//   XtsTransport/XtsTransport Instance <-> NC-Task 1/Axes/Mover Axis 86
//     PlcTask Inputs/GVL_XTS.AxisRefMover[86].NcToPlc <-> Outputs/ToPlc
//     PlcTask Outputs/GVL_XTS.AxisRefMover[86].PlcToNc <-> Inputs/FromPlc
//   XtsTransport/XtsTransport Instance <-> NC-Task 1/Axes/Mover Axis 87
//     PlcTask Inputs/GVL_XTS.AxisRefMover[87].NcToPlc <-> Outputs/ToPlc
//     PlcTask Outputs/GVL_XTS.AxisRefMover[87].PlcToNc <-> Inputs/FromPlc
//   XtsTransport/XtsTransport Instance <-> NC-Task 1/Axes/Mover Axis 88
//     PlcTask Inputs/GVL_XTS.AxisRefMover[88].NcToPlc <-> Outputs/ToPlc
//     PlcTask Outputs/GVL_XTS.AxisRefMover[88].PlcToNc <-> Inputs/FromPlc
//   XtsTransport/XtsTransport Instance <-> NC-Task 1/Axes/Mover Axis 89
//     PlcTask Inputs/GVL_XTS.AxisRefMover[89].NcToPlc <-> Outputs/ToPlc
//     PlcTask Outputs/GVL_XTS.AxisRefMover[89].PlcToNc <-> Inputs/FromPlc
//   XtsTransport/XtsTransport Instance <-> NC-Task 1/Axes/Mover Axis 9
//     PlcTask Inputs/GVL_XTS.AxisRefMover[9].NcToPlc <-> Outputs/ToPlc
//     PlcTask Outputs/GVL_XTS.AxisRefMover[9].PlcToNc <-> Inputs/FromPlc
//   XtsTransport/XtsTransport Instance <-> NC-Task 1/Axes/Mover Axis 90
//     PlcTask Inputs/GVL_XTS.AxisRefMover[90].NcToPlc <-> Outputs/ToPlc
//     PlcTask Outputs/GVL_XTS.AxisRefMover[90].PlcToNc <-> Inputs/FromPlc
//   XtsTransport/XtsTransport Instance <-> NC-Task 1/Axes/Mover Axis 91
//     PlcTask Inputs/GVL_XTS.AxisRefMover[91].NcToPlc <-> Outputs/ToPlc
//     PlcTask Outputs/GVL_XTS.AxisRefMover[91].PlcToNc <-> Inputs/FromPlc
//   XtsTransport/XtsTransport Instance <-> NC-Task 1/Axes/Mover Axis 92
//     PlcTask Inputs/GVL_XTS.AxisRefMover[92].NcToPlc <-> Outputs/ToPlc
//     PlcTask Outputs/GVL_XTS.AxisRefMover[92].PlcToNc <-> Inputs/FromPlc
//   XtsTransport/XtsTransport Instance <-> NC-Task 1/Axes/Mover Axis 93
//     PlcTask Inputs/GVL_XTS.AxisRefMover[93].NcToPlc <-> Outputs/ToPlc
//     PlcTask Outputs/GVL_XTS.AxisRefMover[93].PlcToNc <-> Inputs/FromPlc
//   XtsTransport/XtsTransport Instance <-> NC-Task 1/Axes/Mover Axis 94
//     PlcTask Inputs/GVL_XTS.AxisRefMover[94].NcToPlc <-> Outputs/ToPlc
//     PlcTask Outputs/GVL_XTS.AxisRefMover[94].PlcToNc <-> Inputs/FromPlc
//   XtsTransport/XtsTransport Instance <-> NC-Task 1/Axes/Mover Axis 95
//     PlcTask Inputs/GVL_XTS.AxisRefMover[95].NcToPlc <-> Outputs/ToPlc
//     PlcTask Outputs/GVL_XTS.AxisRefMover[95].PlcToNc <-> Inputs/FromPlc
//   XtsTransport/XtsTransport Instance <-> NC-Task 1/Axes/Mover Axis 96
//     PlcTask Inputs/GVL_XTS.AxisRefMover[96].NcToPlc <-> Outputs/ToPlc
//     PlcTask Outputs/GVL_XTS.AxisRefMover[96].PlcToNc <-> Inputs/FromPlc
//   XtsTransport/XtsTransport Instance <-> NC-Task 1/Axes/Mover Axis 97
//     PlcTask Inputs/GVL_XTS.AxisRefMover[97].NcToPlc <-> Outputs/ToPlc
//     PlcTask Outputs/GVL_XTS.AxisRefMover[97].PlcToNc <-> Inputs/FromPlc
//   XtsTransport/XtsTransport Instance <-> NC-Task 1/Axes/Mover Axis 98
//     PlcTask Inputs/GVL_XTS.AxisRefMover[98].NcToPlc <-> Outputs/ToPlc
//     PlcTask Outputs/GVL_XTS.AxisRefMover[98].PlcToNc <-> Inputs/FromPlc
//   XtsTransport/XtsTransport Instance <-> NC-Task 1/Axes/Mover Axis 99
//     PlcTask Inputs/GVL_XTS.AxisRefMover[99].NcToPlc <-> Outputs/ToPlc
//     PlcTask Outputs/GVL_XTS.AxisRefMover[99].PlcToNc <-> Inputs/FromPlc
//   XtsTransport/XtsTransport Instance <-> NC-Task 1/Objects/Group1 (CA Group)
//     PlcTask Inputs/GVL_XTS.CaGroupRef.NcToPlc/CA <-> Group Outputs/ToPLC
//     PlcTask Outputs/GVL_XTS.CaGroupRef.PlcToNc/CA <-> Group Inputs/FromPLC

// ---- APPLICATION/_types/E_PROCESS_CTRL.TcDUT
{attribute 'qualified_only'}
{attribute 'strict'}
{attribute 'to_string'}
TYPE E_PROCESS_CTRL :
(
  PROCESS_INIT              := 10,
  PROCESS_DISABLE           := 20,
  PROCESS_ENABLE            := 30,

  PROCESS_STATIONS_ENTER    := 40,
  PROCESS_STATIONS_SEND,

  PROCESS_START             := 60,
  PROCESS_DONE              := 70,
  PROCESS_STATIONS_OUTFEED  := 80
);
END_TYPE

// ---- APPLICATION/_types/LinkedList/ST_PROCESS_LIST_RESULT.TcDUT
TYPE ST_PROCESS_LIST_RESULT :
STRUCT
  wState    : WORD;   // wState == 0 --> all ok
  nIndex    : ULINT;
  stData    : ST_PROCESS_DATA;  // copy of list entry
END_STRUCT
END_TYPE

// ---- MAPPING/_types/U_APP_CTRL.TcDUT
TYPE U_APP_CTRL :
UNION
  stCtrl              : ST_APP_CTRL;
  byCtrl    AT %Q*    : ARRAY[1..SIZEOF(ST_APP_CTRL)] OF BYTE;
END_UNION
END_TYPE

// ---- XTS_TRANSPORT/XtsStation/types/E_STATION_GEAR_DISTANCE_AXIS.TcDUT
{attribute 'qualified_only'}
{attribute 'strict'}
{attribute 'to_string'}
TYPE E_STATION_GEAR_DISTANCE_AXIS :
(
  // which axis nSync distance is checked for termination of GearInPosCA.
  // after nSync distance the station does a regular outfeed to target station
	FOLLOW_THE_MASTER,
  FOLLOW_THE_SLAVE
)UINT;
END_TYPE

// ---- _MSG/types/ST_MESSAGE_STATE.TcDUT
TYPE ST_MESSAGE_STATE :
STRUCT
  State         : E_MESSAGE_STATE;  // as always... combined value of Cmd equivalent and e_progress
END_STRUCT
END_TYPE

// ---- APPLICATION/GVL_APPLICATION.TcGVL
VAR_GLOBAL CONSTANT
  MAX_PROCESS       : UINT := 20;
END_VAR
{attribute 'qualified_only'}
VAR_GLOBAL
  Simulation        : ARRAY[1..MAX_PROCESS] OF fb_Simulation;
END_VAR

// ---- XTS_TRANSPORT/GVL_XTS_CONSTANTS.TcGVL
//{attribute 'qualified_only'}
VAR_GLOBAL CONSTANT
//-----------------------------------------------------------------------------------------------------------------------------------------
//-----------------------------------------------------------------------------------------------------------------------------------------
//
//  HAUD 2026.03.15
//  - parameter list deleted (never used the parameter feature anyway), 
//    back to static global constants
//
//-----------------------------------------------------------------------------------------------------------------------------------------
//-----------------------------------------------------------------------------------------------------------------------------------------
//  Connections to XTS Utility Lib data: 
//  - suits this simple approach, 
//  - leaves you options to expand, 
//  - expansion and multiplication is not implemented here on purpose, 
//  - this project is designed to get the main ideas across, 
//  - setting up a matrix for multiple fb_Xpu instances with it, 
//    --> a second step you might want to organize from here; 
//        --> I leave the details up to you
//-----------------------------------------------------------------------------------------------------------------------------------------
//-----------------------------------------------------------------------------------------------------------------------------------------
  MAX_MOVER             : UINT    := 108;
//   MAX_MOVER           : UINT    := TO_UINT(Tc3_XTS_Utility.TcIoXtsEnvironmentParameterList.MaxXtsMoversPerXpu);
//   MAX_MODULE          : UINT    := TO_UINT(Tc3_XTS_Utility.TcIoXtsEnvironmentParameterList.MaxModulesPerPart);
//   MAX_PART            : UINT    := TO_UINT(Tc3_XTS_Utility.TcIoXtsEnvironmentParameterList.MaxXtsPartsPerXpu);
//   MAX_TRACK           : UINT    := TO_UINT(Tc3_XTS_Utility.TcIoXtsEnvironmentParameterList.MaxXtsTracksPerXpu);
//   MAX_GROUP           : UINT    := TO_UINT(Tc3_XTS_Utility.TcIoXtsEnvironmentParameterList.MaxXtsCaGroup);
// 
//   MAX_INFO_SERVER     : UINT    := TO_UINT(Tc3_XTS_Utility.TcIoXtsEnvironmentParameterList.MaxXtsInfoServer);
//   MAX_INFO_STATION    : UINT    := TO_UINT(Tc3_XTS_Utility.TcIoXtsEnvironmentParameterList.MaxXtsInfoStation);
//   MAX_INFO_STOP_POS   : UINT    := TO_UINT(Tc3_XTS_Utility.TcIoXtsEnvironmentParameterList.MaxXtsStopPositionsPerStation);
// 
//   MAX_PARAMETER_SET   : UINT    := TO_UINT(Tc3_XTS_Utility.TcIoXtsEnvironmentParameterList.MaxXtsParameterSet);
// 
//   MAX_NCT_BASE_UNIT   : UINT    := TO_UINT(Tc3_XTS_Utility.TcIoXtsEnvironmentParameterList.MaxXtsNctBaseUnitInterfaces);
//-----------------------------------------------------------------------------------------------------------------------------------------
//-----------------------------------------------------------------------------------------------------------------------------------------
//  XTS_TRANSPORT_LAYER
//  - project constants you will have to adjust in order to build your transport logic
//-----------------------------------------------------------------------------------------------------------------------------------------
//-----------------------------------------------------------------------------------------------------------------------------------------
  MAX_STATION         : UINT    := 150;

  MAX_STATION_NEST    : UINT    := TO_UINT(SIZEOF(ST_STATION_STATE.nMask)*8);
  MAX_LIST_NODES      : UINT    := MAX_MOVER;
  MAX_MASTER          : UINT    := 1;
//-----------------------------------------------------------------------------------------------------------------------------------------
//-----------------------------------------------------------------------------------------------------------------------------------------
END_VAR

// ---- XTS_TRANSPORT/GVL_XTS_VERSION.TcGVL
{attribute 'qualified_only'}
VAR_GLOBAL CONSTANT
//-----------------------------------------------------------------------------------
//-----------------------------------------------------------------------------------
// HAUD 2026 07 26
//
//    XTS_TRANSPORT_LAYER project
//    
//    MIT License
//    
//    Copyright (c) 2025 HAUD
//    
//    Permission is hereby granted, free of charge, to any person obtaining a copy
//    of this software and associated documentation files (the "Software"), to deal
//    in the Software without restriction, including without limitation the rights
//    to use, copy, modify, merge, publish, distribute, sublicense, and/or sell
//    copies of the Software, and to permit persons to whom the Software is
//    furnished to do so, subject to the following conditions:
//    
//    The above copyright notice and this permission notice shall be included in all
//    copies or substantial portions of the Software.
//    
//    THE SOFTWARE IS PROVIDED "AS IS", WITHOUT WARRANTY OF ANY KIND, EXPRESS OR
//    IMPLIED, INCLUDING BUT NOT LIMITED TO THE WARRANTIES OF MERCHANTABILITY,
//    FITNESS FOR A PARTICULAR PURPOSE AND NONINFRINGEMENT. IN NO EVENT SHALL THE
//    AUTHORS OR COPYRIGHT HOLDERS BE LIABLE FOR ANY CLAIM, DAMAGES OR OTHER
//    LIABILITY, WHETHER IN AN ACTION OF CONTRACT, TORT OR OTHERWISE, ARISING FROM,
//    OUT OF OR IN CONNECTION WITH THE SOFTWARE OR THE USE OR OTHER DEALINGS IN THE
//    SOFTWARE.
//-----------------------------------------------------------------------------------
  Version             : STRING  := '4.02.18';
//-----------------------------------------------------------------------------------
END_VAR

// ---- _MSG/GVL_MSG_AXIS.TcGVL
{attribute 'qualified_only'}
VAR_GLOBAL CONSTANT
  //-----------------------------------------------------------------------------
  // file paths for message system
  //  - compiler define option WIN switches to Windows file paths
  //-----------------------------------------------------------------------------
{IF defined (WIN)}
  {info 'PLC_MOTION_LAYER: WIN'}
  LOG_DIR               : STRING  := 'C:\TwinCAT\#MsgFiles\';
{ELSE}
  {info 'PLC_MOTION_LAYER: BSD'}
  LOG_DIR               : STRING  := '/usr/local/etc/TwinCAT/#MsgFiles/';
{END_IF}

  LOG_FILE              : STRING  := concat(TO_STRING(TwinCAT_SystemInfoVarList._AppInfo.AdsPort), '_MSG_PLC_');
  LOG_FILE_METRIC       : STRING  := concat(TO_STRING(TwinCAT_SystemInfoVarList._AppInfo.AdsPort), '_MSG_Metrics_');
END_VAR
VAR_GLOBAL
  //-----------------------------------------------------------------------------
  // Message System
  //  - Everybody uses f_MessageSet(ST_Message)
  //    - DECISION WHICH LIST IS MADE IN f_MessageSet !!
  //    - which list to use is determined by e_Device in your message
  //
  //  - MessageData instances are self sufficient and need only 
  //    datafield assignment for correct data-flow
  //
  //
  //-----------------------------------------------------------------------------
  //-----------------------------------------------------------------------------
  //-----------------------------------------------------------------------------
  // (ST_Message.eDevice := from Device_Null to XfcAxis)
  //-----------------------------------------------------------------------------
  MotionMessageData               : fb_MessageDataCtrl;
  MotionMessageCtrl               : st_message_ctrl;
  MotionMessageState              : st_message_state;

  MotionMessages                  : ARRAY[1..GVL_MSG_XTS.MAX_MESSAGE] OF ST_Message;
  MessageMotionIndex              : UINT := 0; // message index for base layer
  MessageMotionError              : UINT := 0; // error counter for base layer
  //-----------------------------------------------------------------------------
  //-----------------------------------------------------------------------------
  // (ST_Message.eDevice := e_Device.Metrics)
  //-----------------------------------------------------------------------------
  MetricMessageData               : fb_MessageDataCtrl;
  MetricMessageCtrl               : st_message_ctrl;
  MetricMessageState              : st_message_state;

  MetricMessages                  : ARRAY[1..GVL_MSG_XTS.MAX_MESSAGE] OF ST_Message;
  MessageMetricIndex              : UINT := 0; // message index for metrics data
  MessageMetricError              : UINT := 0; // error counter for metrics data
  //-----------------------------------------------------------------------------
  //-----------------------------------------------------------------------------
  fbLocalTime                     : fb_LocalTime;
  dtLocalTime                     : DT;
  sLocalTime                      : STRING;
  //-----------------------------------------------------------------------------
  //-----------------------------------------------------------------------------
  //-----------------------------------------------------------------------------
  //-----------------------------------------------------------------------------
{IF defined (TEST)}
  {info 'TEST logging enabled'}
  MessageLevel                    : E_MessageType := eMessageverbose; // a lot of messages
{ELSE}
  MessageLevel                    : E_MessageType := eMessageEmpty; // only errors are written into list 
{END_IF}

  MessageLevelAxisPtp             : ARRAY[1..PLC_CONSTANT.MAX_AXIS]   OF E_MessageType;
  MessageLevelAxisCam             : ARRAY[1..PLC_CONSTANT.MAX_AXIS]   OF E_MessageType;
  MessageLevelAxisFly             : ARRAY[1..PLC_CONSTANT.MAX_AXIS]   OF E_MessageType;
  MessageLevelNciChn              : ARRAY[1..PLC_CONSTANT.MAX_NCI_CH] OF E_MessageType;

  MessageLevelTriggerBox          : ARRAY[1..PLC_CONSTANT.MAX_TRIGGER_BOX]  OF E_MessageType;
  MessageLevelTouchProbe          : ARRAY[1..PLC_CONSTANT.MAX_TOUCH_PROBE]  OF E_MessageType;


  // diag data
  dbg_AxisIdxGearIn               : ARRAY[1..PLC_CONSTANT.MAX_AXIS]      OF BYTE; // diag for Axis gear in
  dbg_AxisIdxGearInMultiMaster    : ARRAY[1..PLC_CONSTANT.MAX_AXIS,1..4] OF BYTE; // diag for Axis gear in multi master
  dbg_AxisIdxCamIn                : ARRAY[1..PLC_CONSTANT.MAX_AXIS]      OF BYTE; // diag for Axis cam in
END_VAR

// ---- _MSG/GVL_MSG_XTS.TcGVL
{attribute 'qualified_only'}
VAR_GLOBAL CONSTANT
  //-----------------------------------------------------------------------------
  // file paths for message system
  //  - compiler define option WIN switches to Windows file paths
  //-----------------------------------------------------------------------------
{IF defined (WIN)}
  {info 'WIN folders'}
  LOG_DIR               : STRING  := 'C:\TwinCAT\#MsgFiles\';       // delimiter at the end is mandatory!!
  CON_DIR               : STRING  := 'C:\TwinCAT\#Configuration\';  // delimiter at the end is mandatory!!
{ELSE}
  {info 'BSD folders'}
  LOG_DIR               : STRING  := '/usr/local/etc/TwinCAT/#MsgFiles/';       // delimiter at the end is mandatory!!
  CON_DIR               : STRING  := '/usr/local/etc/TwinCAT/#Configuration/';  // delimiter at the end is mandatory!!
{END_IF}

  LOG_FILE              : STRING  := 'MSG_XtsTransport_';
  LOG_FILE_APP          : STRING  := 'MSG_Application_';
  LOG_FILE_METRIC       : STRING  := 'MSG_XtsTransportMetrics_';

  MAX_MESSAGE           : UINT    := 2000; // max entry in message list
END_VAR
VAR_GLOBAL
  //-----------------------------------------------------------------------------
  // Message System
  //  - Everybody uses f_MessageSet(ST_Message)
  //    - DECISION WHICH LIST IS MADE IN f_MessageSet !!
  //    - which list to use is determined by e_Device in your message
  //
  //  - MessageData instances are self sufficient and need only 
  //    datafield assignment for correct data-flow
  //
  //
  //-----------------------------------------------------------------------------
  //-----------------------------------------------------------------------------
  //-----------------------------------------------------------------------------
  // (ST_Message.eDevice := e_Device.Application)
  //----------------------------------------------------------------------------- 
  ApplicationMessageData          : fb_MessageDataCtrl;
  ApplicationMessageCtrl          : st_message_ctrl;
  ApplicationMessageState         : st_message_state;

  ApplicationMessages             : ARRAY[1..MAX_MESSAGE] OF ST_Message;
  MessageApplicationIndex         : UINT := 0; // message index for higher layers (grouping, Instances, etc.)
  MessageApplicationError         : UINT := 0; // error counter for higher learning
  //-----------------------------------------------------------------------------
  //-----------------------------------------------------------------------------
  // (ST_Message.eDevice := from Device_Null to XfcAxis)
  //-----------------------------------------------------------------------------
  TransportMessageData            : fb_MessageDataCtrl;
  TransportMessageCtrl            : st_message_ctrl;
  TransportMessageState           : st_message_state;

  TransportMessages               : ARRAY[1..MAX_MESSAGE] OF ST_Message;
  MessageTransportIndex           : UINT := 0; // message index for base layer
  MessageTransportError           : UINT := 0; // error counter for base layer
  //-----------------------------------------------------------------------------
  //-----------------------------------------------------------------------------
  // (ST_Message.eDevice := e_Device.Metrics)
  //-----------------------------------------------------------------------------
  MetricsMessageData              : fb_MessageDataCtrl;
  MetricsMessageCtrl              : st_message_ctrl;
  MetricsMessageState             : st_message_state;

  MetricsMessages                 : ARRAY[1..MAX_MESSAGE] OF ST_Message;
  MessageMetricsIndex             : UINT := 0; // message index for metrics data
  MessageMetricsError             : UINT := 0; // error counter for metrics data
  //-----------------------------------------------------------------------------
  //-----------------------------------------------------------------------------
  // (ST_Message.eDevice := e_Device.ProductData)
  //-----------------------------------------------------------------------------
  ProductMessageData              : fb_MessageDataCtrl;   // This is for you
  ProductMessageCtrl              : st_message_ctrl;
  ProductMessageState             : st_message_state;

  ProductMessages                 : ARRAY[1..MAX_MESSAGE] OF ST_Message;
  MessageProductIndex             : UINT := 0; // message index for your product data
  MessageProductError             : UINT := 0; // error counter for your product data
  //-----------------------------------------------------------------------------
  //-----------------------------------------------------------------------------
  fbLocalTime                     : fb_LocalTime;
  dtLocalTime                     : DT;
  sLocalTime                      : STRING;
  //-----------------------------------------------------------------------------
  //-----------------------------------------------------------------------------
  //-----------------------------------------------------------------------------
  //-----------------------------------------------------------------------------
  MessageLevelXpu                 : E_MessageType;
  MessageLevelStations            : ARRAY[1..MAX_STATION] OF E_MessageType;
  MessageLevelMovers              : ARRAY[1..MAX_MOVER]   OF E_MessageType;

  MessageLevelProcess             : ARRAY[1..MAX_PROCESS] OF E_MessageType;

{IF defined (TEST)}
  {info 'TEST logging enabled'}
  MessageLevel                    : E_MessageType := eMessageinfo; // a lot of messages
{ELSE}
  MessageLevel                    : E_MessageType := eMessageEmpty; // only errors are written into list 
{END_IF}

END_VAR

// ---- APPLICATION/fb_Simulation.TcPOU
//---------------------------------------------------------------------------------------------------------------
//
//  HAUD 2023.03.27
//
//
//  fb_Simulation
//
//    !!! NOT FOR USE IN PRODUCTION !!! --> build something from your mind, this gets messy if you do not
//
//  - grouping of xts stations to sync start process
//  - nFirst to nLast xts stations are checked for starting process simultaneously
//  - basic preparation of station target index in PrepareTarget()
//  - handshake with station control for mover transport through station
//
//---------------------------------------------------------------------------------------------------------------
// This SOFTWARE is provided as an Exemple by THE PROVIDER "as is" and "with all faults." THE PROVIDER makes no 
// representations or warranties of any kind concerning the safety, suitability, lack of viruses, inaccuracies, 
// typographical errors, or other harmful components of this SOFTWARE. There are inherent dangers in the use of 
// any software, and you are solely responsible for determining whether this SOFTWARE is compatible with your 
// equipment and other software installed on your equipment. You are also solely responsible for the protection 
// of your equipment and backup of your data, and THE PROVIDER will not be liable for any damages you may suffer 
// in connection with using, modifying, or distributing this SOFTWARE.
//---------------------------------------------------------------------------------------------------------------
FUNCTION_BLOCK fb_Simulation
VAR
  _nProcessId                 : UINT;

  _sCheck                     : STRING;
  _tonProcess                 : Tc2_Standard.TON;
  _tProcess                   : TIME := T#500MS;

  _AllStationMoverPerMinute   : UDINT;
  _nMoverCountTotal           : UDINT;

  _tonPartsPerMinute          : Tc2_Standard.TON;

  {attribute 'displaymode':='bin'}
  _wEnter                     : DWORD;
  {attribute 'displaymode':='bin'}
  _wStart                     : DWORD;
  {attribute 'displaymode':='bin'}
  _wOut                       : DWORD;
  {attribute 'displaymode':='bin'}
  _wGone                      : DWORD;
  {attribute 'displaymode':='bin'}
  _wEnableProcess             : DWORD; // bits switch on stations

  {attribute 'displaymode':='bin'}
  _TargetMask                 : BYTE;

  _stCtrl                     : POINTER TO ARRAY[1..MAX_STATION]  OF ST_STATION_CTRL;
  _stState                    : POINTER TO ARRAY[1..MAX_STATION]  OF ST_STATION_STATE;

  // controlling bits from properties used on the outside
  _bNext,
  _bMoverEnter,
  _bMoverOut                  : BOOL;

  // who is included in process
  // _nFirst to _nLast MUST be in closed consecutive order
  _nProcessState,
  _nStation,
  _nStationCount,
  _nFirstStation,
  _nLastStation               : UINT;

  _nTarget,
  _nFirstTarget,
  _nLastTarget                : UINT;

  _nPreparedTarget            : ARRAY[1..MAX_MOVER]  OF UINT;

  _nMoverCountStartOld,
  _nMoverCountEnterOld,
  _nMoverCountEnter,
  _nMoverCountStart,
  _nMoverPerMinute,
  _nMoverCount,
  _nMoverCountOld             : ARRAY[1..MAX_STATION]  OF UDINT;

  _rCheckRangeLow,
  _rCheckRangeHigh            : LREAL; // position range the mover has to be in for infeed or sending to happen.

  _MessageLevel               : E_MessageType;
  _stMsg                      : ST_Message;
END_VAR

METHOD Check : BOOL

IF (_nFirstStation < 1) OR
   (_nFirstStation > MAX_STATION)
THEN
  _sCheck                     := '_nFirstStation out of bounds';
  RETURN;
END_IF

IF (_nLastStation < 1) OR
   (_nLastStation > MAX_STATION)
THEN
  _sCheck                     := '_nLastStation out of bounds';
  RETURN;
END_IF

IF (_nFirstTarget < 1) OR
   (_nFirstTarget > MAX_STATION)
THEN
  _sCheck                     := '_nFirstTarget out of bounds';
  RETURN;
END_IF

IF (_nLastTarget < 1) OR
   (_nLastTarget > MAX_STATION)
THEN
  _sCheck                     := '_nLastTarget out of bounds';
  RETURN;
END_IF

IF NOT (_stCtrl  <> 0)
THEN
  _sCheck                     := '_stCtrl: missing pointer';
  RETURN;
END_IF

IF NOT (_stState <> 0)
THEN
  _sCheck                     := '_stState: missing pointer';
  RETURN;
END_IF


_sCheck                       := TO_STRING(E_PROGRESS.PROGRESS_DONE);
Check                         := TRUE;
END_METHOD

PROPERTY CheckRangeHigh : lreal
GET
CheckRangeHigh := _rCheckRangeHigh;
END_GET
SET
_rCheckRangeHigh := CheckRangeHigh;
END_SET
END_PROPERTY

PROPERTY CheckRangeLow : lreal
GET
CheckRangeLow := _rCheckRangeLow;
END_GET
SET
_rCheckRangeLow := CheckRangeLow;
END_SET
END_PROPERTY

METHOD Cycle
VAR_INST
  _interAllStationsCounter    : UDINT;

  _rtrigProcessEnter,
  _rtrigProcessStart,
  _rtrigProcess       : ARRAY[1..MAX_STATION] OF Tc2_Standard.R_TRIG;

  _k                  : UINT;
  _wEnable            : DWORD;
END_VAR
//-----------------------------------------------------------------------------------------------------------------
IF NOT Check() THEN RETURN; END_IF
//-----------------------------------------------------------------------------------------------------------------
_nStationCount                              := _nLastStation - _nFirstStation + 1;
//-----------------------------------------------------------------------------------------------------------------
//-----------------------------------------------------------------------------------------------------------------
IF (_nStationCount < 1)
THEN
  RETURN;
END_IF
//-----------------------------------------------------------------------------------------------------------------
//-----------------------------------------------------------------------------------------------------------------
FOR _nStation := _nLastStation TO _nFirstStation BY(-1) 
DO
  CASE _stState^[_nStation].State
  OF
    //-------------------------------------------------------------------------------------------------------------
    E_STATION_STATE.STATION_DISABLE,
    E_STATION_STATE.STATION_ENABLE, 
    E_STATION_STATE.STATION_DETECT_MOVER:
      _wStart   := _wOut    := _wGone       := 0;
      _wEnter                               := DelBit(_wEnter, (_nStation-_nFirstStation));
      IF (GetBit(_wEnableProcess, (_nStation-_nFirstStation)))
      THEN
        IF (_bMoverEnter)
        THEN
          _stCtrl^[_nStation].Cmd           := E_STATION_CTRL.STATION_ENABLE;
        ELSE
          _stCtrl^[_nStation].Cmd           := E_STATION_CTRL.STATION_DISABLE;
        END_IF
      ELSE
        _stCtrl^[_nStation].Cmd             := E_STATION_CTRL.STATION_DISABLE;
      END_IF


    //-------------------------------------------------------------------------------------------------------------
    E_STATION_STATE.STATION_MOVER_ENTER:
      _wEnter                               := SetBit(_wEnter, (_nStation-_nFirstStation));
      IF _bMoverEnter
      THEN
        _tonProcess(IN                      := FALSE, 
                    PT                      := _tProcess);

        _stCtrl^[_nStation].nTargetStation  := 0;

        IF (_tProcess < T#10MS)
        THEN
          IF (_rCheckRangeHigh > _rCheckRangeLow)
          THEN
            IF (_stState^[_nStation].rMoverModPos > _rCheckRangeLow) AND
               (_stState^[_nStation].rMoverModPos < _rCheckRangeHigh)
            THEN
              _stCtrl^[_nStation].Cmd       := E_STATION_CTRL.STATION_MOVER_SEND;
            END_IF
          ELSE
            IF (_stState^[_nStation].rMoverModPos > _rCheckRangeLow) OR
               (_stState^[_nStation].rMoverModPos < _rCheckRangeHigh)
            THEN
              _stCtrl^[_nStation].Cmd       := E_STATION_CTRL.STATION_MOVER_SEND;
            END_IF
          END_IF
        ELSE
          IF (_rCheckRangeHigh > _rCheckRangeLow)
          THEN
            IF (_stState^[_nStation].rMoverModPos > _rCheckRangeLow) AND
               (_stState^[_nStation].rMoverModPos < _rCheckRangeHigh)
            THEN
              _stCtrl^[_nStation].Cmd       := E_STATION_CTRL.STATION_MOVER_ENTER;
            END_IF
          ELSE
            IF (_stState^[_nStation].rMoverModPos > _rCheckRangeLow) OR
               (_stState^[_nStation].rMoverModPos < _rCheckRangeHigh)
            THEN
              _stCtrl^[_nStation].Cmd       := E_STATION_CTRL.STATION_MOVER_ENTER;
            END_IF
          END_IF
        END_IF
      END_IF

    //-------------------------------------------------------------------------------------------------------------
    E_STATION_STATE.STATION_PROCESS_START:
      _wEnter                               := DelBit(_wEnter, (_nStation-_nFirstStation));
      _wStart                               := SetBit(_wStart, (_nStation-_nFirstStation));
  
      // check if ALL XtsStations have mover in place to work
      IF (_wStart = _wEnableProcess)
      THEN
        _tonProcess(IN                      := TRUE, 
                    PT                      := _tProcess);

        IF _tonProcess.Q
        THEN
          PrepareTargets(FALSE);
          _stCtrl^[_nStation].Cmd           := E_STATION_CTRL.STATION_PROCESS_DONE;
        END_IF
      END_IF

    //-------------------------------------------------------------------------------------------------------------
    E_STATION_STATE.STATION_CHECK_NEST:
      _wEnter                               := SetBit(_wEnter, (_nStation-_nFirstStation));
      _wStart                               := DelBit(_wStart, (_nStation-_nFirstStation));
      _tonProcess(IN                        := FALSE, 
                  PT                        := _tProcess);

      IF (_bNext)
      THEN
        // check if ALL XtsStations have nest to work
        IF (_wEnter = _wEnableProcess)
        THEN
          _stCtrl^[_nStation].Cmd           := E_STATION_CTRL.STATION_MOVER_ENTER;
        END_IF
      END_IF

    //-------------------------------------------------------------------------------------------------------------
    E_STATION_STATE.STATION_MOVER_OUT:
      _wOut                                 := SetBit(_wOut, (_nStation-_nFirstStation));
      _tonProcess(IN                        := FALSE, 
                  PT                        := _tProcess);

      IF _bMoverOut
      THEN
        // nest mask for this mover in target station, sender decides what to work in target
        _stCtrl^[_nStation].nMask           := _TargetMask;

        // check if ALL XtsStations have mover to send
        IF (_wOut = _wEnableProcess)
        THEN
          _nProcessState                    := 10;
        END_IF
      END_IF
  END_CASE
END_FOR
//-----------------------------------------------------------------------------------------------------------------
//-----------------------------------------------------------------------------------------------------------------
CASE _nProcessState
OF
10:
  // ctrl has to decide where to send mover; this depends on YOUR decision
  IF PrepareTargets(TRUE)
  THEN
    PrepareTargets(FALSE);
    _nProcessState                          := 30;
  END_IF
END_CASE
CASE _nProcessState
OF
30:
  FOR _nStation := _nLastStation TO _nFirstStation BY(-1) 
  DO
    IF _bNext
    THEN
      // start outfeed of mover
      _stCtrl^[_nStation].Cmd               := E_STATION_CTRL.STATION_MOVER_OUT;
    END_IF

    CASE _stState^[_nStation].State
    OF
      E_STATION_STATE.STATION_MOVER_GONE:
        _wStart   := _wEnter                := 0;
        // whO is gone?
        _wGone                              := SetBit(_wGone, (_nStation-_nFirstStation));
    END_CASE
  END_FOR
  // check if ALL XtsStations are empty
  IF (_wGone = _wEnableProcess)
  THEN
    _nProcessState                          := 40;
    IF (_MessageLevel > E_MessageType.eMessageVerbose)
    THEN
      _stMsg.eType                          := E_MessageType.eMessageSentient;
      _stMsg.eDevice                        := e_Device.MetricsXts + TO_UINT(_nProcessId);
      _stMsg.eSubdevice                     := e_Subdevice.Process_StationCollector;
      _stMsg.iErrorNumber                   := _nProcessId;
      _stMsg.sText                          := concat('ALL MOVER: ', TO_STRING(E_STATION_STATE.STATION_MOVER_GONE));

      f_MessageSet(_stMsg);
    END_IF
  END_IF
END_CASE
CASE _nProcessState
OF
40:
  _nProcessState                            := 0;
  FOR _nStation := _nLastStation TO _nFirstStation BY(-1) 
  DO
    // let XtsStations jump back to disable
    _stCtrl^[_nStation].Cmd                 := E_STATION_CTRL.STATION_MOVER_GONE;
  END_FOR
END_CASE
//-----------------------------------------------------------------------------------------------------------------
//-----------------------------------------------------------------------------------------------------------------
//-----------------------------------------------------------------------------------------------------------------
// Mover per Minute counter all XtsStations in range
//-----------------------------------------------------------------------------------------------------------------
_nMoverCountTotal                           :=
_AllStationMoverPerMinute                   := 0; 
//-----------------------------------------------------------------------------------------------------------------
// mover counter
//-----------------------------------------------------------------------------------------------------------------
FOR _k := _nLastStation TO _nFirstStation BY(-1)
DO
  //---------------------------------------------------------------------------------------------------------------
  _rtrigProcess[_k](CLK:= ( _stCtrl^[_k].Cmd = E_STATION_CTRL.STATION_MOVER_OUT));
  //---------------------------------------------------------------------------------------------------------------
  IF _rtrigProcess[_k].Q
  THEN
    _nMoverCount[_k]                        := _nMoverCount[_k] + 1;

    IF (_MessageLevel > E_MessageType.eMessageError)
    THEN
      _stMsg.eType                          := E_MessageType.eMessageInfo;
      _stMsg.eDevice                        := e_Device.MetricsXts + TO_UINT(_nProcessId);
      _stMsg.eSubdevice                     := e_Subdevice.Process_StationCollector;
      _stMsg.iErrorNumber                   := _k;
      _stMsg.sText                          := concat('MoverCountStation[ ]: ', TO_STRING(_nMoverCount[_k]));
      _stMsg.sText                          := concat(_stMsg.sText, ': E_STATION_CTRL.');
      _stMsg.sText                          := concat(_stMsg.sText, TO_STRING(_stCtrl^[_k].Cmd));
      f_MessageSet(_stMsg);
    END_IF
  END_IF

  //---------------------------------------------------------------------------------------------------------------
  _rtrigProcessStart[_k](CLK:= ( _stState^[_k].State = E_STATION_STATE.STATION_PROCESS_START));
  //---------------------------------------------------------------------------------------------------------------
  IF _rtrigProcessStart[_k].Q
  THEN
    _nMoverCountStart[_k]                   := _nMoverCountStart[_k] + 1;

    IF (_MessageLevel > E_MessageType.eMessageInfo)
    THEN
      _stMsg.eType                          := E_MessageType.eMessageVerbose;
      _stMsg.eDevice                        := e_Device.MetricsXts + TO_UINT(_nProcessId);
                            
      _stMsg.eSubdevice                     := e_Subdevice.Process_StationCollector;
      _stMsg.iErrorNumber                   := _k;
      _stMsg.sText                          := concat('MoverCountStation[ ]: ', TO_STRING(_nMoverCountEnter[_k]));
      _stMsg.sText                          := concat(_stMsg.sText, ': E_STATION_STATE.');
      _stMsg.sText                          := concat(_stMsg.sText, TO_STRING(_stState^[_k].State));
      f_MessageSet(_stMsg);
    END_IF
  END_IF

  //---------------------------------------------------------------------------------------------------------------
  _rtrigProcessEnter[_k](CLK:= ( _stCtrl^[_k].Cmd = E_STATION_CTRL.STATION_MOVER_ENTER));
  //---------------------------------------------------------------------------------------------------------------
  IF _rtrigProcessEnter[_k].Q
  THEN
    _nMoverCountEnter[_k]                   := _nMoverCountEnter[_k] + 1;

    IF (_MessageLevel > E_MessageType.eMessageVerbose)
    THEN
      _stMsg.eType                          := E_MessageType.eMessageSentient;
      _stMsg.eDevice                        := e_Device.MetricsXts + TO_UINT(_nProcessId);
                            
      _stMsg.eSubdevice                     := e_Subdevice.Process_StationCollector;
      _stMsg.iErrorNumber                   := _k;
      _stMsg.sText                          := concat('MoverCountStation[ ]: ', TO_STRING(_nMoverCountEnter[_k]));
      _stMsg.sText                          := concat(_stMsg.sText, ': E_STATION_CTRL.');
      _stMsg.sText                          := concat(_stMsg.sText, TO_STRING(_stCtrl^[_k].Cmd));
      f_MessageSet(_stMsg);
    END_IF
  END_IF
  //---------------------------------------------------------------------------------------------------------------
  //---------------------------------------------------------------------------------------------------------------
  IF _tonPartsperMinute.Q
  THEN
    // count every XtsStation in range
    _nMoverPerMinute[_k]                    := _nMoverCount[_k] - _nMoverCountOld[_k];
    _nMoverCountOld [_k]                    := _nMoverCount[_k];

    _nMoverCountEnterOld [_k]               := _nMoverCountEnter[_k];
    _nMoverCountStartOld [_k]               := _nMoverCountStart[_k];
  END_IF
  // sum up all XtsStations in range
  _AllStationMoverPerMinute                 := _AllStationMoverPerMinute + _nMoverPerMinute[_k]; 
  _interAllStationsCounter                  := _AllStationMoverPerMinute + _nMoverPerMinute[_k];

  // sum up all mover counts in range
  _nMoverCountTotal                         := _nMoverCountTotal + _nMoverCount[_k];
END_FOR
//-----------------------------------------------------------------------------------------------------------------
//-----------------------------------------------------------------------------------------------------------------
// total mover per minute message for all stations in this process
//-----------------------------------------------------------------------------------------------------------------
//-----------------------------------------------------------------------------------------------------------------
IF _tonPartsperMinute.q
THEN
  _tonPartsperMinute(IN:=FALSE);

  IF (_MessageLevel > E_MessageType.eMessageError)
  THEN
    _stMsg.eType                          := E_MessageType.eMessageBatch;
    _stMsg.eDevice                        := e_Device.MetricsXts + TO_UINT(_nProcessId);
  
    _stMsg.eSubdevice                     := e_Subdevice.Process_StationCollector;
    _stMsg.iErrorNumber                   := _nMoverCountTotal;
    _stMsg.sText                          := concat('MoverCountTotal: ', TO_STRING(_nMoverCountTotal));
    _stMsg.sText                          := concat(_stMsg.sText, ': StationLast: ');
    _stMsg.sText                          := concat(_stMsg.sText, TO_STRING(_nLastStation));
    _stMsg.sText                          := concat(_stMsg.sText, ': StationFirst: ');
    _stMsg.sText                          := concat(_stMsg.sText, TO_STRING(_nFirstStation));
    f_MessageSet(_stMsg);
  END_IF
END_IF
//-----------------------------------------------------------------------------------------------------------------
_tonPartsperMinute(IN:= TRUE,   PT:= T#60S);
//-----------------------------------------------------------------------------------------------------------------
//-----------------------------------------------------------------------------------------------------------------
END_METHOD

METHOD PUBLIC DelBit : DWORD
VAR_INPUT
  inVal   : DWORD;
  bitNo   : DINT;
END_VAR
VAR
  wConst : dWORD := 1;
END_VAR
IF ( inVal AND SHL( wConst,bitNo MOD 32 ) ) > 0 THEN
  DelBit := inVal XOR (SHL( wConst,bitNo MOD 32 ));
ELSE
  DelBit := inVal;
END_IF
END_METHOD

METHOD Disable : BOOL
VAR_INPUT
END_VAR
IF NOT (_nLastStation   > 0) OR
   NOT (_nFirstStation  > 0) OR
   NOT (_nLastStation   < MAX_STATION+1) OR
   NOT (_nFirstStation  < MAX_STATION+1)
THEN
  Disable := FALSE;
ELSE
  FOR _nStation := _nLastStation TO _nFirstStation BY(-1) 
  DO
    _stCtrl^[_nStation].Cmd               := E_STATION_CTRL.STATION_DISABLE;
    _stCtrl^[_nStation].nMask             := 0;
  END_FOR

  memset(ADR(_nMoverCount),    0, SIZEOF(_nMoverCount));
  memset(ADR(_nMoverCountOld), 0, SIZEOF(_nMoverCountOld));
  _nProcessState :=  _nTarget             := 0;
  
  Disable := TRUE;
END_IF
END_METHOD

PROPERTY EnableProcess : dword
GET
EnableProcess := _wEnableProcess;
END_GET
SET
_wEnableProcess := EnableProcess;
END_SET
END_PROPERTY

METHOD PUBLIC GetBit : BOOL
VAR_INPUT
  inVal   : DWORD;
  bitNo   : DINT;
END_VAR
VAR
  wConst : DWORD := 1;
END_VAR
IF ( inVal AND SHL( wConst,DINT_TO_SINT(bitNo) MOD 32 ) ) > 0
THEN
  GetBit := TRUE;
ELSE
  GetBit := FALSE;
END_IF
END_METHOD

METHOD Init : BOOL
VAR_INPUT
END_VAR
IF NOT (_nLastStation   > 0) OR
   NOT (_nFirstStation  > 0) OR
   NOT (_nLastStation   < MAX_STATION+1) OR
   NOT (_nFirstStation  < MAX_STATION+1)
THEN
  Init := FALSE;
ELSE
  FOR _nStation := _nLastStation TO _nFirstStation BY(-1) 
  DO
    _stCtrl^[_nStation].Cmd               := E_STATION_CTRL.STATION_INIT;
    _stCtrl^[_nStation].nMask             := 0;
  END_FOR

  memset(ADR(_nMoverCount),    0, SIZEOF(_nMoverCount));
  memset(ADR(_nMoverCountOld), 0, SIZEOF(_nMoverCountOld));
  _nProcessState :=  _nTarget             := 0;
  
  Init := TRUE;
END_IF
END_METHOD

PROPERTY MessageLevel : e_MessageType
GET
MessageLevel := _MessageLevel;
END_GET
SET
VAR
  _ix : uint;
END_VAR
_MessageLevel := MessageLevel;
END_SET
END_PROPERTY

PROPERTY MoverEnter : bool
GET
MoverEnter := _bMoverEnter;
END_GET
SET
_bMoverEnter := MoverEnter;
END_SET
END_PROPERTY

PROPERTY MoverOut : bool
GET
MoverOut := _bMoverOut;
END_GET
SET
_bMoverOut := MoverOut;
END_SET
END_PROPERTY

METHOD Next : BOOL
VAR_INPUT
  Nxt  : Bool;
END_VAR
_bNext := Nxt;
END_METHOD

METHOD PRIVATE PrepareTargets : BOOL
VAR_INPUT
  Execute         : BOOL;
END_VAR
VAR_INST
  _idxStations    : uint;
  _nt,
  _nstate         : UINT;
END_VAR

IF NOT Check() THEN RETURN; END_IF

IF NOT Execute
THEN
  _nstate                             := 0;
END_IF


CASE _nstate
OF
  0:
    IF Execute
    THEN
      _nstate                         := 10;
    END_IF
END_CASE
CASE _nstate
OF
  10:
    _nstate                           := 20;

    FOR _idxStations := _nLastStation TO _nFirstStation BY(-1) 
    DO
      _nt                               := TO_USINT(_nLastTarget - _nTarget);
      _nTarget                          := _nTarget + 1;
  
      _nPreparedTarget[_stState^[_idxStations].nMoverId]  := _nt;
      _stCtrl^[_idxStations].nTargetStation               := TO_USINT(_nt);
  
      IF (_nLastTarget - _nTarget < _nFirstTarget)
      THEN
        _nTarget                        := 0;
      END_IF
    END_FOR
END_CASE
CASE _nstate
OF
  20:
    PrepareTargets                    := TRUE;
END_CASE
END_METHOD

PROPERTY ProcessId : uint
GET
ProcessId := _nProcessId;
END_GET
SET
_nProcessId := ProcessId;
END_SET
END_PROPERTY

PROPERTY ProcessTime : time
GET
ProcessTime := _tProcess;
END_GET
SET
_tProcess := ProcessTime;
END_SET
END_PROPERTY

METHOD PUBLIC SetBit : DWORD
VAR_INPUT
  inVal   : DWORD;
  bitNo   : DINT;
END_VAR
VAR
  wConst  : dWORD := 1;
END_VAR
SetBit := inVal OR SHL( wConst,bitNo MOD 32 );
END_METHOD

PROPERTY StationCount : uint
GET
StationCount := _nStationCount;
END_GET
END_PROPERTY

PROPERTY StationCtrl : pointer to ARRAY[1..MAX_STATION]  OF ST_STATION_CTRL;
SET
_stCtrl := StationCtrl;
END_SET
END_PROPERTY

PROPERTY StationFirst : uint
GET
StationFirst := _nFirstStation;
END_GET
SET
_nFirstStation := StationFirst;
END_SET
END_PROPERTY

PROPERTY StationLast : uint
GET
StationLast := _nLastStation;
END_GET
SET
_nLastStation := StationLast;
END_SET
END_PROPERTY

PROPERTY StationState : POINTER TO ARRAY[1..MAX_STATION]  OF ST_STATION_STATE
SET
_stState := StationState;
END_SET
END_PROPERTY

PROPERTY TargetFirst : uint
GET
TargetFirst := _nFirstTarget;
END_GET
SET
_nFirstTarget := TargetFirst;
END_SET
END_PROPERTY

PROPERTY TargetLast : uint
GET
TargetLast := _nLastTarget;
END_GET
SET
_nLastTarget := TargetLast;
END_SET
END_PROPERTY

PROPERTY TargetMask : byte
GET
TargetMask := _TargetMask;
END_GET
SET
_TargetMask := TargetMask;
END_SET
END_PROPERTY

END_FUNCTION_BLOCK

// ---- _MSG/f_MessageSet.TcPOU
FUNCTION f_MessageSet : BOOL
VAR_INPUT
  stMessage     : ST_Message;
END_VAR
VAR
  _uiIndex      : UINT;
  _MainDevice   : e_Device;
  _nModRes      : UDINT;     // residual after modulo
END_VAR

stMessage.tTime                     := GVL_MSG_XTS.sLocalTime;

// why here? so all calls to this function may stay the same
_nModRes                            := stMessage.eDevice MOD e_Device.General;
_MainDevice                         := stMessage.eDevice - _nModRes;

CASE _MainDevice
OF
  //--------------------------------------------------------------------------------
  e_device.DataProduct:
    // this is your data, if you choose to use this message system
    FOR _uiIndex := 1 TO GVL_MSG_XTS.MAX_MESSAGE
    DO
      IF (GVL_MSG_XTS.ProductMessages[_uiIndex].eType = e_MessageType.eMessageEmpty)
      THEN
        GVL_MSG_XTS.ProductMessages[_uiIndex]      := stMessage;
        GVL_MSG_XTS.MessageProductIndex            := _uiIndex;
        EXIT;
      END_IF
    END_FOR
  
    IF (stMessage.eType = E_MessageType.eMessageError)
    THEN
      // in case of error: increment counter
      GVL_MSG_XTS.MessageProductError              := GVL_MSG_XTS.MessageProductError + 1;
    END_IF
  //--------------------------------------------------------------------------------
  e_Device.Process,
  e_Device.Application:
    FOR _uiIndex := 1 TO GVL_MSG_XTS.MAX_MESSAGE
    DO
      IF (GVL_MSG_XTS.ApplicationMessages[_uiIndex].eType = e_MessageType.eMessageEmpty)
      THEN
        GVL_MSG_XTS.ApplicationMessages[_uiIndex]  := stMessage;    // yes, we grab global values directly, only here
        GVL_MSG_XTS.MessageApplicationIndex        := _uiIndex;
        EXIT;
      END_IF
    END_FOR
    IF (stMessage.eType = E_MessageType.eMessageError)
    THEN
      // in case of error: increment counter
      GVL_MSG_XTS.MessageApplicationError          := GVL_MSG_XTS.MessageApplicationError + 1;
    END_IF
  //--------------------------------------------------------------------------------
  e_Device.MetricsXts:
    FOR _uiIndex := 1 TO GVL_MSG_XTS.MAX_MESSAGE
    DO
      IF (GVL_MSG_XTS.MetricsMessages[_uiIndex].eType = e_MessageType.eMessageEmpty)
      THEN
        GVL_MSG_XTS.MetricsMessages[_uiIndex]      := stMessage;    // yes, we grab global values directly, only here
        GVL_MSG_XTS.MessageMetricsIndex            := _uiIndex;
        EXIT;
      END_IF
    END_FOR
    IF (stMessage.eType = E_MessageType.eMessageError)
    THEN
      // in case of error: increment counter
      GVL_MSG_XTS.MessageMetricsError              := GVL_MSG_XTS.MessageMetricsError + 1;
    END_IF
  //--------------------------------------------------------------------------------
  e_Device.MetricsAxis:
    FOR _uiIndex := 1 TO GVL_MSG_XTS.MAX_MESSAGE
    DO
      IF (GVL_MSG_AXIS.MetricMessages[_uiIndex].eType = e_MessageType.eMessageEmpty)
      THEN
        GVL_MSG_AXIS.MetricMessages[_uiIndex]  := stMessage;    // yes, we grab global values directly, only here
        GVL_MSG_AXIS.MessageMetricIndex        := _uiIndex;
        EXIT;
      END_IF
    END_FOR
    IF (stMessage.eType = E_MessageType.eMessageError)
    THEN
      // in case of error: increment counter
      GVL_MSG_AXIS.MessageMetricError          := GVL_MSG_AXIS.MessageMetricError + 1;
    END_IF
  //--------------------------------------------------------------------------------
  e_Device.Axis,
  e_Device.XfcAxis,
  e_device.XfcTouchProbe,
  e_device.XfcTriggerBox,
  e_Device.Camming,
  e_device.NciChannel,
  e_device.NciChannelCtrl:
    FOR _uiIndex := 1 TO GVL_MSG_XTS.MAX_MESSAGE
    DO
      IF (GVL_MSG_AXIS.MotionMessages[_uiIndex].eType = e_MessageType.eMessageEmpty)
      THEN
        GVL_MSG_AXIS.MotionMessages[_uiIndex]  := stMessage;    // yes, we grab global values directly, only here
        GVL_MSG_AXIS.MessageMotionIndex        := _uiIndex;
        EXIT;
      END_IF
    END_FOR
    IF (stMessage.eType = E_MessageType.eMessageError)
    THEN
      // in case of error: increment counter
      GVL_MSG_AXIS.MessageMotionError           := GVL_MSG_AXIS.MessageMotionError + 1;
    END_IF
  //--------------------------------------------------------------------------------
ELSE
  CASE stMessage.eDevice
  OF
    Device_MainApplication,
    Device_XmlData,              
    Device_Utilities:
      FOR _uiIndex := 1 TO GVL_MSG_XTS.MAX_MESSAGE
      DO
        IF (GVL_MSG_XTS.ApplicationMessages[_uiIndex].eType = e_MessageType.eMessageEmpty)
        THEN
          GVL_MSG_XTS.ApplicationMessages[_uiIndex]:= stMessage;    // yes, we grab global values directly, only here
          GVL_MSG_XTS.MessageApplicationIndex      := _uiIndex;
          EXIT;
        END_IF
      END_FOR
      IF (stMessage.eType = E_MessageType.eMessageError)
      THEN
        // in case of error: increment counter
        GVL_MSG_XTS.MessageApplicationError        := GVL_MSG_XTS.MessageApplicationError + 1;
      END_IF

    Device_MainAxis,
    Device_Nci,
    Device_Cam,
    Device_Functions,
    Device_FlyingSaw,
    Device_ParameterSelector:     // PLC_MOTION
      FOR _uiIndex := 1 TO GVL_MSG_XTS.MAX_MESSAGE
      DO
        IF (GVL_MSG_AXIS.MotionMessages[_uiIndex].eType = e_MessageType.eMessageEmpty)
        THEN
          GVL_MSG_AXIS.MotionMessages[_uiIndex]:= stMessage;    // yes, we grab global values directly, only here
          GVL_MSG_AXIS.MessageMotionIndex      := _uiIndex;
          EXIT;
        END_IF
      END_FOR
      IF (stMessage.eType = E_MessageType.eMessageError)
      THEN
        // in case of error: increment counter
        GVL_MSG_AXIS.MessageMotionError        := GVL_MSG_AXIS.MessageMotionError + 1;
      END_IF

    Device_Main,
    Device_MoverSelector:
      FOR _uiIndex := 1 TO GVL_MSG_XTS.MAX_MESSAGE
      DO
        IF (GVL_MSG_XTS.TransportMessages[_uiIndex].eType = e_MessageType.eMessageEmpty)
        THEN
          GVL_MSG_XTS.TransportMessages[_uiIndex]  := stMessage;
          GVL_MSG_XTS.MessageTransportIndex        := _uiIndex;
          EXIT;
        END_IF
      END_FOR
  ELSE    
    //--------------------------------------------------------------------------------
    FOR _uiIndex := 1 TO GVL_MSG_XTS.MAX_MESSAGE
    DO
      IF (GVL_MSG_XTS.TransportMessages[_uiIndex].eType = e_MessageType.eMessageEmpty)
      THEN
        GVL_MSG_XTS.TransportMessages[_uiIndex]    := stMessage;
        GVL_MSG_XTS.MessageTransportIndex          := _uiIndex;
        EXIT;
      END_IF
    END_FOR
  
    IF (stMessage.eType = E_MessageType.eMessageError)
    THEN
      // in case of error: increment counter
      GVL_MSG_XTS.MessageTransportError := GVL_MSG_XTS.MessageTransportError + 1;
    END_IF
  END_CASE
END_CASE

END_FUNCTION

// ---- MAIN.TcPOU
//---------------------------------------------------------------------------------------------------------------
//
//  HAUD 2026.01.16
//
//  - ExternControl
//
//    - placeholder programm for specific implementation of machine logic
//
//---------------------------------------------------------------------------------------------------------------
PROGRAM MAIN
VAR
	bInit 				          : BOOL;
  eInit                   : E_PROGRESS := E_PROGRESS.PROGRESS_DONE; // empty right now, so init is done

  nStation,
	nMover,
  nMoverSelected,
  nStationSelected,
  nStationParameter       : UINT;

  sStationText            : STRING(30);
  stXpuStrings            : ST_XPU_STRINGS;

  eTransportState         : E_XTS_TRANSPORT_STATE;
  eTransportResult        : E_PROGRESS;

  eXpuState               : E_XPU_STATE;
  eXpuResult              : E_PROGRESS;
  eXpuCheck               : E_XPU_CHECK;

  eMoverState             : E_MOVER_STATE;
  eMoverResult            : E_PROGRESS;

  sCaGroupState,
  sTransportState,
  sTransportCheck,
  sTransportResult,
  sMoverState,
  sMoverResult,
  sStationState,
  sStationStateMask,
  sStationCtrlMask        : STRING;

  bStationEnable,
  bStationEnter,
  bStationStart,
  bStationDone,
  bStationOut,
  bStationGone            : BOOL;

  nStn                    : UINT;

  stMsg                   : ST_Message;
  eMsgState               : e_message_state;
  eMsgProgress            : E_PROGRESS;
  eMtrState               : e_message_state;
  eMtrProgress            : E_PROGRESS;

  bGetVariant             : BOOL := TRUE;
  nVariant                : UINT;

  rGap                    : REAL :=     105.0;
  rAcc                    : REAL :=  17_500.0;
  rJerk                   : REAL := 600_000.0;
END_VAR

//############################################################################
//############################################################################
//  /Visualization data	
//############################################################################
VisualizationData();
//############################################################################
//  Visualization data/	
//############################################################################

ACTION VisualizationData:
//############################################################################
//############################################################################
// Visualization data	
//############################################################################
// get enumerations from XPU for visu:	
eTransportState                       := f_GetState   (GVL_XTS.XtsTransportState.State);
eTransportResult                      := f_GetProgress(GVL_XTS.XtsTransportState.State);

eXpuState                             := f_GetState   (GVL_XTS.XtsTransportState.XpuState.State);
eXpuResult                            := f_GetProgress(GVL_XTS.XtsTransportState.XpuState.State);

eXpuCheck                             := GVL_XTS.XtsTransportState.XpuState.Check;

// display xpu state and result in visu
// get strings and info
sCaGroupState                         := TO_STRING(GVL_XTS.XtsTransportState.GroupInfo.CaGroupState);

sTransportState                       := TO_STRING(eTransportState);
sTransportCheck                       := TO_STRING(GVL_XTS.XtsTransportState.Check);
sTransportResult                      := TO_STRING(eTransportResult);

stXpuStrings.sXpuState                := TO_STRING(eXpuState);
stXpuStrings.sXpuResult               := TO_STRING(eXpuResult);
stXpuStrings.sXpuCyclicCheck          := TO_STRING(eXpuCheck);

stXpuStrings.sXpuOpMode               := TO_STRING(GVL_XTS.XtsTransportState.XpuInfo.OperationMode);
stXpuStrings.sXpuMoverId_DetectionMode:= TO_STRING(GVL_XTS.XtsTransportState.XpuInfo.IdDetectionMode);
stXpuStrings.sXpuMoverPosAssignement  := TO_STRING(GVL_XTS.XtsTransportState.XpuInfo.MoverPositionAssignement);

nMoverSelected                        := SEL((nMoverSelected<1), nMoverSelected, 1);
nMoverSelected                        := SEL((nMoverSelected>MAX_MOVER), nMoverSelected, MAX_MOVER);

nStationSelected                      := SEL((nStationSelected<1), nStationSelected, 1);
nStationSelected                      := SEL((nStationSelected>MAX_STATION), nStationSelected, MAX_STATION);

bStationEnable                        := SEL((GVL_XTS.StationCtrl[nStationSelected].Cmd = E_STATION_CTRL.STATION_ENABLE),        FALSE, TRUE);
bStationEnter                         := SEL((GVL_XTS.StationCtrl[nStationSelected].Cmd = E_STATION_CTRL.STATION_MOVER_ENTER),   FALSE, TRUE);
bStationStart                         := SEL((GVL_XTS.StationCtrl[nStationSelected].Cmd = E_STATION_CTRL.STATION_PROCESS_START), FALSE, TRUE);
bStationDone                          := SEL((GVL_XTS.StationCtrl[nStationSelected].Cmd = E_STATION_CTRL.STATION_PROCESS_DONE),  FALSE, TRUE);
bStationOut                           := SEL((GVL_XTS.StationCtrl[nStationSelected].Cmd = E_STATION_CTRL.STATION_MOVER_OUT),     FALSE, TRUE);
bStationGone                          := SEL((GVL_XTS.StationCtrl[nStationSelected].Cmd = E_STATION_CTRL.STATION_MOVER_GONE),    FALSE, TRUE);

eMoverState                           := f_GetState   (GVL_XTS.MoverState[nMoverSelected].State);
eMoverResult                          := f_GetProgress(GVL_XTS.MoverState[nMoverSelected].State);

sMoverState                           := TO_STRING(eMoverState);
sMoverResult                          := TO_STRING(eMoverResult);

sStationState                         := TO_STRING(GVL_XTS.StationState[nStationSelected].State);
sStationStateMask                     := Tc2_Utilities.BYTE_TO_BINSTR(GVL_XTS.StationState[nStationSelected].nMask, 8);
sStationCtrlMask                      := Tc2_Utilities.BYTE_TO_BINSTR(GVL_XTS.StationCtrl[nStationSelected].nMask, 8);

//############################################################################
//############################################################################
END_ACTION

END_PROGRAM

// ---- _types/f_GetProgress.TcPOU
// global function to extract e_progress from combined value
FUNCTION f_GetProgress : uint
VAR_INPUT
  state     : UINT;
END_VAR
VAR
  nP        : uint;
END_VAR


nP := state / E_PROGRESS.PROGRESS_INIT;

f_GetProgress := nP * E_PROGRESS.PROGRESS_INIT;

END_FUNCTION

// ---- APPLICATION/MAIN_APP.TcPOU
//---------------------------------------------------------------------------------------------------------------
//
//  HAUD 2026.01.16
//
//  - ExternControl
//
//    - cyclic call to simulation class which handshakes the XtsStations in XtsTransport PLC
//
//---------------------------------------------------------------------------------------------------------------
PROGRAM MAIN_APP
VAR
  eInitXtsTransport   AT %I*    : e_progress;
  eInit                         : E_PROGRESS;   // application startup state info

  nProcess          : UINT;

  bNext             : BOOL := TRUE;
  bEnter            : BOOL := TRUE;
  bLeave            : BOOL := TRUE;

  tProcess          : ARRAY[1..MAX_PROCESS] OF TIME;

  eMtrState,
  eMsgState         : E_MESSAGE_STATE;
  eMtrProgress,
  eMsgProgress      : e_progress;
  stMsg             : ST_Message;
  //-------------------------------------------------------------------------------------------------------------
  tIdleWriteApplication   : TIME := T#5S;
  tIdleWriteMetric        : TIME := T#5S;
  tonIdleWriteApplication : Tc2_Standard.TON;
  tonIdleWriteMetric      : Tc2_Standard.TON;
  //-------------------------------------------------------------------------------------------------------------
END_VAR

//#################################################################################################################
// Local time; used for timestamps
//#################################################################################################################
GVL_MSG_XTS.fbLocalTime();
GVL_MSG_XTS.sLocalTime                                      := GVL_MSG_XTS.fbLocalTime.LocalTimeString;
GVL_MSG_XTS.dtLocalTime                                     := GVL_MSG_XTS.fbLocalTime.LocalTime;
//#################################################################################################################
//#################################################################################################################
//-----------------------------------------------------------------------------------------------------------------
//-----------------------------------------------------------------------------------------------------------------
// check for MAIN.eInit
//  - wait for fb_TransportUnit to be fully started up
//-----------------------------------------------------------------------------------------------------------------
IF NOT (eInitXtsTransport = E_PROGRESS.PROGRESS_DONE) THEN eInit   := E_PROGRESS.PROGRESS_INVALID; RETURN; END_IF
//-----------------------------------------------------------------------------------------------------------------
//-----------------------------------------------------------------------------------------------------------------
//-----------------------------------------------------------------------------------------------------------------
// /assign dataflow
//-----------------------------------------------------------------------------------------------------------------
FOR nProcess := 1 TO MAX_PROCESS
DO
  GVL_APPLICATION.Simulation[nProcess].ProcessId            := nProcess;
  GVL_APPLICATION.Simulation[nProcess].StationCtrl          := ADR(GVL_XTS.StationCtrl);
  GVL_APPLICATION.Simulation[nProcess].StationState         := ADR(GVL_XTS.StationState);

  GVL_APPLICATION.Simulation[nProcess].ProcessTime          := tProcess[nProcess];
  GVL_APPLICATION.Simulation[nProcess].MessageLevel         := GVL_MSG_XTS.MessageLevel;
END_FOR
//-----------------------------------------------------------------------------------------------------------------
//-----------------------------------------------------------------------------------------------------------------
Init();
//-----------------------------------------------------------------------------------------------------------------
//-----------------------------------------------------------------------------------------------------------------
// react to operation modes
//-----------------------------------------------------------------------------------------------------------------
//-----------------------------------------------------------------------------------------------------------------
CASE GVL_XTS.XtsTransportCtrl.Cmd
OF
  E_XTS_TRANSPORT_CTRL.CMD_INIT,
  E_XTS_TRANSPORT_CTRL.CMD_GROUP_CLEAR:

    FOR nProcess := 1 TO MAX_PROCESS
    DO
      GVL_APPLICATION.Simulation[nProcess].Init(); // clearing of XtsStations and Simulation
    END_FOR
END_CASE

CASE (GVL_XTS.XtsTransportState.State MOD E_PROGRESS.PROGRESS_DONE)
OF
  E_XTS_TRANSPORT_STATE.TRANSPORT_INIT,
  E_XTS_TRANSPORT_STATE.TRANSPORT_GROUP_CLEAR:
    FOR nProcess := 1 TO MAX_PROCESS
    DO
      GVL_APPLICATION.Simulation[nProcess].Disable(); // switch off XtsStations and clear Simulation

      GVL_APPLICATION.Simulation[nProcess].EnableProcess    := 0;
      GVL_APPLICATION.Simulation[nProcess].MoverEnter       := FALSE;
      GVL_APPLICATION.Simulation[nProcess].MoverOut         := FALSE;

      GVL_APPLICATION.Simulation[nProcess].Cycle();
    END_FOR

  E_XTS_TRANSPORT_STATE.TRANSPORT_START,
  E_XTS_TRANSPORT_STATE.TRANSPORT_RESTART:

    FOR nProcess := 1 TO MAX_PROCESS
    DO
      GVL_APPLICATION.Simulation[nProcess].Next(bNext);
      GVL_APPLICATION.Simulation[nProcess].Cycle();
    END_FOR
ELSE
  CASE (GVL_XTS.XtsTransportState.State MOD E_PROGRESS.PROGRESS_WORKING)
  OF
  E_XTS_TRANSPORT_STATE.TRANSPORT_START,
  E_XTS_TRANSPORT_STATE.TRANSPORT_RESTART:
    FOR nProcess := 1 TO MAX_PROCESS
    DO
      IF (GVL_APPLICATION.Simulation[nProcess].StationCount > 0)
      THEN
        GVL_APPLICATION.Simulation[nProcess].EnableProcess  := TO_DWORD(EXPT(2,GVL_APPLICATION.Simulation[nProcess].StationCount))-1;
        GVL_APPLICATION.Simulation[nProcess].MoverEnter     := TRUE;
        GVL_APPLICATION.Simulation[nProcess].MoverOut       := TRUE;

      END_IF

      GVL_APPLICATION.Simulation[nProcess].Next(bNext);
      GVL_APPLICATION.Simulation[nProcess].Cycle();
    END_FOR
  END_CASE
END_CASE
//-----------------------------------------------------------------------------------------------------------------
//-----------------------------------------------------------------------------------------------------------------
//#################################################################################################################
// /logging
//#################################################################################################################
GVL_MSG_XTS.ApplicationMessageData.Ctrl                         REF= GVL_MSG_XTS.ApplicationMessageCtrl;
GVL_MSG_XTS.ApplicationMessageData.State                        REF= GVL_MSG_XTS.ApplicationMessageState;

GVL_MSG_XTS.ApplicationMessageData.MessageIndex                 REF= GVL_MSG_XTS.MessageApplicationIndex;
GVL_MSG_XTS.ApplicationMessageData.ErrorIndex                   REF= GVL_MSG_XTS.MessageApplicationError;

GVL_MSG_XTS.ApplicationMessageData.DirRoot                      :=   ADR(GVL_MSG_XTS.LOG_DIR);
GVL_MSG_XTS.ApplicationMessageData.FileRoot                     :=   ADR(GVL_MSG_XTS.LOG_FILE_APP);
GVL_MSG_XTS.ApplicationMessageData.MsgList                      :=   ADR(GVL_MSG_XTS.ApplicationMessages);
GVL_MSG_XTS.ApplicationMessageData.LocalTime                    :=   ADR(GVL_MSG_XTS.dtLocalTime);

GVL_MSG_XTS.ApplicationMessageData();

eMsgState                                   := f_GetState   (GVL_MSG_XTS.ApplicationMessageState.State);
eMsgProgress                                := f_GetProgress(GVL_MSG_XTS.ApplicationMessageState.State);


CASE eMsgState
OF
  E_MESSAGE_STATE.MSG_STATE_NULL:
    CASE eMsgProgress
    OF
      E_PROGRESS.PROGRESS_INVALID:
        IF (GVL_MSG_XTS.MessageApplicationIndex > GVL_MSG_XTS.MAX_MESSAGE/100) OR
           (GVL_MSG_XTS.MessageApplicationError > 0)
        THEN
          GVL_MSG_XTS.ApplicationMessageCtrl.Cmd  := E_MESSAGE_CTRL.MSG_CTRL_WRITE;
        ELSE
          tonIdleWriteApplication(IN := TRUE, PT:= tIdleWriteApplication);
          IF (tonIdleWriteApplication.Q)
          THEN
            GVL_MSG_XTS.TransportMessageCtrl.Cmd    := E_MESSAGE_CTRL.MSG_CTRL_WRITE;
          END_IF
        END_IF
    END_CASE

  E_MESSAGE_STATE.MSG_STATE_WRITE:
    CASE eMsgProgress
    OF
      E_PROGRESS.PROGRESS_ERROR,
      E_PROGRESS.PROGRESS_DONE:
        tonIdleWriteApplication(IN := FALSE, PT:= tIdleWriteApplication);
        GVL_MSG_XTS.ApplicationMessageCtrl.Cmd    := E_MESSAGE_CTRL.MSG_CTRL_NULL;
    END_CASE

ELSE
    CASE eMsgProgress
    OF
      E_PROGRESS.PROGRESS_DONE:
        GVL_MSG_XTS.ApplicationMessageCtrl.Cmd    := E_MESSAGE_CTRL.MSG_CTRL_NULL;
    END_CASE
END_CASE
//#################################################################################################################
// logging/
//#################################################################################################################
//#################################################################################################################
//  /Transport Metrics
//#################################################################################################################
GVL_MSG_XTS.MetricsMessageData.Ctrl                             REF= GVL_MSG_XTS.MetricsMessageCtrl;
GVL_MSG_XTS.MetricsMessageData.State                            REF= GVL_MSG_XTS.MetricsMessageState;

GVL_MSG_XTS.MetricsMessageData.MessageIndex                     REF= GVL_MSG_XTS.MessageMetricsIndex;
GVL_MSG_XTS.MetricsMessageData.ErrorIndex                       REF= GVL_MSG_XTS.MessageMetricsError;

GVL_MSG_XTS.MetricsMessageData.DirRoot                          :=   ADR(GVL_MSG_XTS.LOG_DIR);
GVL_MSG_XTS.MetricsMessageData.FileRoot                         :=   ADR(GVL_MSG_XTS.LOG_FILE_METRIC);
GVL_MSG_XTS.MetricsMessageData.MsgList                          :=   ADR(GVL_MSG_XTS.MetricsMessages);
GVL_MSG_XTS.MetricsMessageData.LocalTime                        :=   ADR(GVL_MSG_XTS.dtLocalTime);

GVL_MSG_XTS.MetricsMessageData();

eMtrState                                   := f_GetState   (GVL_MSG_XTS.MetricsMessageState.State);
eMtrProgress                                := f_GetProgress(GVL_MSG_XTS.MetricsMessageState.State);

CASE eMtrState
OF
  E_MESSAGE_STATE.MSG_STATE_NULL:
    CASE eMtrProgress
    OF
      E_PROGRESS.PROGRESS_INVALID:
        IF (GVL_MSG_XTS.MessageMetricsIndex > GVL_MSG_XTS.MAX_MESSAGE/100) OR
           (GVL_MSG_XTS.MessageMetricsError > 0)
        THEN
          GVL_MSG_XTS.MetricsMessageCtrl.Cmd      := E_MESSAGE_CTRL.MSG_CTRL_WRITE;
        ELSE
          tonIdleWriteMetric(IN := TRUE, PT:= tIdleWriteMetric);
          IF (tonIdleWriteMetric.Q)
          THEN
            GVL_MSG_XTS.TransportMessageCtrl.Cmd    := E_MESSAGE_CTRL.MSG_CTRL_WRITE;
          END_IF
        END_IF
    END_CASE

  E_MESSAGE_STATE.MSG_STATE_WRITE:
    CASE eMtrProgress
    OF
      E_PROGRESS.PROGRESS_ERROR,
      E_PROGRESS.PROGRESS_DONE:
        tonIdleWriteMetric(IN := FALSE, PT:= tIdleWriteMetric);
        GVL_MSG_XTS.MetricsMessageCtrl.Cmd        := E_MESSAGE_CTRL.MSG_CTRL_NULL;
    END_CASE
ELSE
    CASE eMtrProgress
    OF
      E_PROGRESS.PROGRESS_DONE:
        GVL_MSG_XTS.MetricsMessageCtrl.Cmd        := E_MESSAGE_CTRL.MSG_CTRL_NULL;
    END_CASE
END_CASE
//#################################################################################################################
//  Transport Metrics/
//#################################################################################################################
//#################################################################################################################
//#################################################################################################################

ACTION Init:
CASE eInit
OF
  E_PROGRESS.PROGRESS_INVALID:          // startup procedure for your application
    GVL_MSG_XTS.TransportMessageCtrl.Cmd                  := E_MESSAGE_CTRL.MSG_CTRL_NULL;
    GVL_MSG_XTS.MetricsMessageCtrl.Cmd                    := E_MESSAGE_CTRL.MSG_CTRL_NULL;

    FOR nProcess := 1 TO MAX_PROCESS
    DO
      GVL_MSG_XTS.MessageLevelProcess[nProcess]           := GVL_MSG_XTS.MessageLevel;

      GVL_APPLICATION.Simulation[nProcess].MessageLevel   := GVL_MSG_XTS.MessageLevelProcess[nProcess];
    END_FOR
    eInit                               := E_PROGRESS.PROGRESS_INIT;


  E_PROGRESS.PROGRESS_INIT:
      nProcess                                        := 1;
      tProcess[nProcess]                              := T#750MS;

      GVL_APPLICATION.Simulation[nProcess].StationFirst  := 1;
      GVL_APPLICATION.Simulation[nProcess].StationLast   := 16;

      GVL_APPLICATION.Simulation[nProcess].TargetFirst   := 20;
      GVL_APPLICATION.Simulation[nProcess].TargetLast    := 35;
      GVL_APPLICATION.Simulation[nProcess].TargetMask    := 2#0001; // mask for target station

      GVL_APPLICATION.Simulation[nProcess].CheckRangeLow := 1750.0;
      GVL_APPLICATION.Simulation[nProcess].CheckRangeHigh:= 2100.0;

      //---------------------------------------------------------

      // 2

      //---------------------------------------------------------
      nProcess                                        := 3;
      tProcess[nProcess]                              := T#1250MS;

      GVL_APPLICATION.Simulation[nProcess].StationFirst  := 20;
      GVL_APPLICATION.Simulation[nProcess].StationLast   := 35;

      GVL_APPLICATION.Simulation[nProcess].TargetFirst   := 37;
      GVL_APPLICATION.Simulation[nProcess].TargetLast    := 37;
      GVL_APPLICATION.Simulation[nProcess].TargetMask    := 2#0001; // mask for target station

      GVL_APPLICATION.Simulation[nProcess].CheckRangeLow := 4500.0;
      GVL_APPLICATION.Simulation[nProcess].CheckRangeHigh:= 5100.0;

      //---------------------------------------------------------
      nProcess                                        := 4;
      tProcess[nProcess]                              := T#0MS;

      GVL_APPLICATION.Simulation[nProcess].StationFirst  := 37;
      GVL_APPLICATION.Simulation[nProcess].StationLast   := 37;

      GVL_APPLICATION.Simulation[nProcess].TargetFirst   := 45;
      GVL_APPLICATION.Simulation[nProcess].TargetLast    := 52;
      GVL_APPLICATION.Simulation[nProcess].TargetMask    := 2#0001; // mask for target station

      GVL_APPLICATION.Simulation[nProcess].CheckRangeLow := 7450.0;
      GVL_APPLICATION.Simulation[nProcess].CheckRangeHigh:= 7600.0;

      //---------------------------------------------------------
      nProcess                                        := 5;
      tProcess[nProcess]                              := T#500MS;

      GVL_APPLICATION.Simulation[nProcess].StationFirst  := 45;
      GVL_APPLICATION.Simulation[nProcess].StationLast   := 52;

      GVL_APPLICATION.Simulation[nProcess].TargetFirst   := 58;
      GVL_APPLICATION.Simulation[nProcess].TargetLast    := 69;
      GVL_APPLICATION.Simulation[nProcess].TargetMask    := 2#0001; // mask for target station

      GVL_APPLICATION.Simulation[nProcess].CheckRangeLow := 6600.0;
      GVL_APPLICATION.Simulation[nProcess].CheckRangeHigh:= 8350.0;

      //---------------------------------------------------------
      nProcess                                        := 6;
      tProcess[nProcess]                              := T#500MS;

      GVL_APPLICATION.Simulation[nProcess].StationFirst  := 58;
      GVL_APPLICATION.Simulation[nProcess].StationLast   := 69;

      GVL_APPLICATION.Simulation[nProcess].TargetFirst   := 70;
      GVL_APPLICATION.Simulation[nProcess].TargetLast    := 81;
      GVL_APPLICATION.Simulation[nProcess].TargetMask    := 2#0001; // mask for target station

      GVL_APPLICATION.Simulation[nProcess].CheckRangeLow := 8750.0;
      GVL_APPLICATION.Simulation[nProcess].CheckRangeHigh:= 9600.0;

      //---------------------------------------------------------
      nProcess                                        := 7;
      tProcess[nProcess]                              := T#500MS;

      GVL_APPLICATION.Simulation[nProcess].StationFirst  := 70;
      GVL_APPLICATION.Simulation[nProcess].StationLast   := 81;

      GVL_APPLICATION.Simulation[nProcess].TargetFirst   := 82;
      GVL_APPLICATION.Simulation[nProcess].TargetLast    := 91;
      GVL_APPLICATION.Simulation[nProcess].TargetMask    := 2#0001; // mask for target station

      GVL_APPLICATION.Simulation[nProcess].CheckRangeLow := 10900.0;
      GVL_APPLICATION.Simulation[nProcess].CheckRangeHigh:= 11600.0;

      //---------------------------------------------------------
      nProcess                                        := 8;
      tProcess[nProcess]                              := T#500MS;

      GVL_APPLICATION.Simulation[nProcess].StationFirst  := 82;
      GVL_APPLICATION.Simulation[nProcess].StationLast   := 91;

      GVL_APPLICATION.Simulation[nProcess].TargetFirst   := 92;
      GVL_APPLICATION.Simulation[nProcess].TargetLast    := 99;
      GVL_APPLICATION.Simulation[nProcess].TargetMask    := 2#0001; // mask for target station

      GVL_APPLICATION.Simulation[nProcess].CheckRangeLow := 12550.0;
      GVL_APPLICATION.Simulation[nProcess].CheckRangeHigh:= 12900.0;

      //---------------------------------------------------------
      nProcess                                        := 9;
      tProcess[nProcess]                              := T#500MS;

      GVL_APPLICATION.Simulation[nProcess].StationFirst  := 92;
      GVL_APPLICATION.Simulation[nProcess].StationLast   := 99;

      GVL_APPLICATION.Simulation[nProcess].TargetFirst   := 118;
      GVL_APPLICATION.Simulation[nProcess].TargetLast    := 118;
      GVL_APPLICATION.Simulation[nProcess].TargetMask    := 2#0001; // mask for target station

      GVL_APPLICATION.Simulation[nProcess].CheckRangeLow := 13600.0;
      GVL_APPLICATION.Simulation[nProcess].CheckRangeHigh:= 14600.0;

      //---------------------------------------------------------
      nProcess                                        := 12;
      tProcess[nProcess]                              := T#600MS;

      GVL_APPLICATION.Simulation[nProcess].StationFirst  := 110;
      GVL_APPLICATION.Simulation[nProcess].StationLast   := 117;

      GVL_APPLICATION.Simulation[nProcess].TargetFirst   := 134;
      GVL_APPLICATION.Simulation[nProcess].TargetLast    := 147;
      GVL_APPLICATION.Simulation[nProcess].TargetMask    := 2#0001; // mask for target station

      GVL_APPLICATION.Simulation[nProcess].CheckRangeLow := 16500.0;
      GVL_APPLICATION.Simulation[nProcess].CheckRangeHigh:= 17100.0;

      //---------------------------------------------------------
      nProcess                                        := 13;
      tProcess[nProcess]                              := T#00MS;

      GVL_APPLICATION.Simulation[nProcess].StationFirst  := 118;
      GVL_APPLICATION.Simulation[nProcess].StationLast   := 118;

      GVL_APPLICATION.Simulation[nProcess].TargetFirst   := 119;
      GVL_APPLICATION.Simulation[nProcess].TargetLast    := 119;
      GVL_APPLICATION.Simulation[nProcess].TargetMask    := 2#0001; // mask for target station

      GVL_APPLICATION.Simulation[nProcess].CheckRangeLow := 15400.0;
      GVL_APPLICATION.Simulation[nProcess].CheckRangeHigh:= 15600.0;

      //---------------------------------------------------------
      nProcess                                        := 14;
      tProcess[nProcess]                              := T#0MS;

      GVL_APPLICATION.Simulation[nProcess].StationFirst  := 119;
      GVL_APPLICATION.Simulation[nProcess].StationLast   := 119;

      GVL_APPLICATION.Simulation[nProcess].TargetFirst   := 110;
      GVL_APPLICATION.Simulation[nProcess].TargetLast    := 117;
      GVL_APPLICATION.Simulation[nProcess].TargetMask    := 2#0001; // mask for target station

      GVL_APPLICATION.Simulation[nProcess].CheckRangeLow := 15750.0;
      GVL_APPLICATION.Simulation[nProcess].CheckRangeHigh:= 16250.0;

      //---------------------------------------------------------


      //---------------------------------------------------------
      nProcess                                        := 16;
      tProcess[nProcess]                              := T#750MS;

      GVL_APPLICATION.Simulation[nProcess].StationFirst  := 134;
      GVL_APPLICATION.Simulation[nProcess].StationLast   := 147;

      GVL_APPLICATION.Simulation[nProcess].TargetFirst   := 148;
      GVL_APPLICATION.Simulation[nProcess].TargetLast    := 148;
      GVL_APPLICATION.Simulation[nProcess].TargetMask    := 2#0001; // mask for target station

      GVL_APPLICATION.Simulation[nProcess].CheckRangeLow := 18500.0;
      GVL_APPLICATION.Simulation[nProcess].CheckRangeHigh:= 19600.0;

      //---------------------------------------------------------
      nProcess                                        := 17;
      tProcess[nProcess]                              := T#0MS;

      GVL_APPLICATION.Simulation[nProcess].StationFirst  := 148;
      GVL_APPLICATION.Simulation[nProcess].StationLast   := 148;

      GVL_APPLICATION.Simulation[nProcess].TargetFirst   := 149;
      GVL_APPLICATION.Simulation[nProcess].TargetLast    := 149;
      GVL_APPLICATION.Simulation[nProcess].TargetMask    := 2#0001; // mask for target station

      GVL_APPLICATION.Simulation[nProcess].CheckRangeLow := 21750.0;
      GVL_APPLICATION.Simulation[nProcess].CheckRangeHigh:= 22100.0;

      //---------------------------------------------------------
      nProcess                                        := 18;
      tProcess[nProcess]                              := T#0MS;

      GVL_APPLICATION.Simulation[nProcess].StationFirst  := 149;
      GVL_APPLICATION.Simulation[nProcess].StationLast   := 149;

      GVL_APPLICATION.Simulation[nProcess].TargetFirst   := 150;
      GVL_APPLICATION.Simulation[nProcess].TargetLast    := 150;
      GVL_APPLICATION.Simulation[nProcess].TargetMask    := 2#0001; // mask for target station

      GVL_APPLICATION.Simulation[nProcess].CheckRangeLow := 22450.0;
      GVL_APPLICATION.Simulation[nProcess].CheckRangeHigh:= 22700.0;

      //---------------------------------------------------------
      nProcess                                        := 19;
      tProcess[nProcess]                              := T#0MS;

      GVL_APPLICATION.Simulation[nProcess].StationFirst  := 150;
      GVL_APPLICATION.Simulation[nProcess].StationLast   := 150;

      GVL_APPLICATION.Simulation[nProcess].TargetFirst   := 1;
      GVL_APPLICATION.Simulation[nProcess].TargetLast    := 16;
      GVL_APPLICATION.Simulation[nProcess].TargetMask    := 2#0001; // mask for target station

      GVL_APPLICATION.Simulation[nProcess].CheckRangeLow := 500.0;
      GVL_APPLICATION.Simulation[nProcess].CheckRangeHigh:= 2100.0;

    eInit                                                 := E_PROGRESS.PROGRESS_BUSY;

  E_PROGRESS.PROGRESS_BUSY:
    GVL_MSG_XTS.TransportMessageCtrl.Cmd                  := E_MESSAGE_CTRL.MSG_CTRL_INIT;
    GVL_MSG_XTS.MetricsMessageCtrl.Cmd                    := E_MESSAGE_CTRL.MSG_CTRL_INIT;
    eInit                                                 := E_PROGRESS.PROGRESS_PREPARE;

  E_PROGRESS.PROGRESS_PREPARE:
    eInit                                                 := E_PROGRESS.PROGRESS_DONE;

END_CASE
END_ACTION

END_PROGRAM

// ---- APPLICATION/_types/fb_Instance/fb_Instance.TcPOU
//---------------------------------------------------------------------------------------------------------------
//
//  HAUD 2024.11.21
//
//
//  fb_Instance
//  - base class for process instance to work with fb_ProcessCollector
//  - basic check and var names, so you can build your procedures with it
//  - processes are connected via linked list
//
//  - inherit this base class for your application, call Check() cyclic
//
//---------------------------------------------------------------------------------------------------------------//
// This SOFTWARE is provided as an Exemple by THE PROVIDER "as is" and "with all faults." THE PROVIDER makes no  //
// representations or warranties of any kind concerning the safety, suitability, lack of viruses, inaccuracies,  //
// typographical errors, or other harmful components of this SOFTWARE. There are inherent dangers in the use of  //
// any software, and you are solely responsible for determining whether this SOFTWARE is compatible with your    //
// equipment and other software installed on your equipment. You are also solely responsible for the protection  //
// of your equipment and backup of your data, and THE PROVIDER will not be liable for any damages you may suffer //
// in connection with using, modifying, or distributing this SOFTWARE.                                           //
//---------------------------------------------------------------------------------------------------------------//
FUNCTION_BLOCK fb_Instance
VAR
  _eState                 : E_INSTANCE_STATE;  // local state machine for infeed procedure
  _eStateProgress         : E_PROGRESS; // substate for lacal state machine

  _eInit                  : E_PROGRESS;
  _eCheck                 : E_INSTANCE_CHECK;  // pointer checks

  // XTS station range
  _nStationLast           : UINT;
  _nStationFirst          : UINT;

  // process index
  _nProcess               : UINT;

  // local ctrl / state datafields for you to use
  _Ctrl                   : ST_PROCESS_CTRL;   // control to write, connected by reference to _ItfProcessCollector
  _State                  : ST_PROCESS_STATE;  // state   to read,  connected by reference to _ItfProcessCollector

  _ItfProcessCollector    : ARRAY[1..MAX_PROCESS] OF I_ProcessCollector;

  _ItfProcessList         : ARRAY[1..MAX_PROCESS] OF I_Process_LinkedList;  // access to all linked lists for process entry
  _ListResult             : ST_PROCESS_LIST_RESULT;
  _ProcessData            : ST_PROCESS_DATA;

  {attribute 'displaymode':='bin'}
  _wTargetUsed            : T_PROCESS;  // bits use XtsStation in target process
  _wTargetMask            : ARRAY[1..SIZEOF(T_PROCESS)*8] OF BYTE;

  _stMsg                  : ST_Message;
  _MessageLevel           : E_MessageType;
END_VAR

METHOD Check : BOOL // call this method in the extending/inheriting class
//-----------------------------------------------------------------------------
//-----------------------------------------------------------------------------
// plausibility checks
//-----------------------------------------------------------------------------
IF NOT (_nProcess > 0)
THEN
  _eCheck                 := E_INSTANCE_CHECK.INVALID_PROCESS_ID_ZERO;
  RETURN;
END_IF

IF NOT (_nProcess < MAX_PROCESS+1)
THEN
  _eCheck                 := E_INSTANCE_CHECK.INVALID_PROCESS_ID_MAX;
  RETURN;
END_IF
//-----------------------------------------------------------------------------
//-----------------------------------------------------------------------------
// pointer checks
//-----------------------------------------------------------------------------
IF NOT (_ItfProcessCollector[_nProcess] <> 0) 
THEN
  _eCheck                 := E_INSTANCE_CHECK.INVALID_INTERFACE_POINTER;
  RETURN;
END_IF

IF NOT (_ItfProcessCollector[_nProcess].ProcessId > 0)
THEN
  _eCheck                 := E_INSTANCE_CHECK.INVALID_PROCESS_ID_ZERO;
  RETURN;
END_IF

IF NOT (_ItfProcessCollector[_nProcess].ProcessId < MAX_PROCESS+1)
THEN
  _eCheck                 := E_INSTANCE_CHECK.INVALID_PROCESS_ID_MAX;
  RETURN;
END_IF

IF NOT (_nProcess = _ItfProcessCollector[_nProcess].ProcessId)
THEN
  _eCheck                 := E_INSTANCE_CHECK.INVALID_PROCESS_ID_NOTEQUAL_COLLECTOR_ID;
  RETURN;
END_IF

IF NOT (_ItfProcessList[_nProcess] <> 0)
THEN
  _eCheck                 := E_INSTANCE_CHECK.INVALID_INDEX_IN_LIST;
  RETURN;
END_IF
//-----------------------------------------------------------------------------
//-----------------------------------------------------------------------------
// connect datafields to interface of ProcessCollector
//-----------------------------------------------------------------------------
_ItfProcessCollector[_nProcess].ProcessCtrl      REF= _Ctrl;
_ItfProcessCollector[_nProcess].ProcessState     REF= _State;
//-----------------------------------------------------------------------------
//-----------------------------------------------------------------------------
// DEBUG: copy station range
//-----------------------------------------------------------------------------
_nStationLast                         := _ItfProcessCollector[_nProcess].StationLast;
_nStationFirst                        := _ItfProcessCollector[_nProcess].StationFirst;
//-----------------------------------------------------------------------------
//-----------------------------------------------------------------------------
// set message device
//-----------------------------------------------------------------------------
_stMsg.eDevice                        := e_Device.Process + _nProcess;
//-----------------------------------------------------------------------------
//-----------------------------------------------------------------------------
_eCheck                   := E_INSTANCE_CHECK.CHECK_DONE;
Check                     := TRUE;
END_METHOD

PROPERTY ProcessId : uint
GET
ProcessId := _nProcess;
END_GET
SET
_nProcess := ProcessId;
END_SET
END_PROPERTY

PROPERTY ProcessInterface : array[1..MAX_PROCESS] of I_ProcessCollector
SET
_ItfProcessCollector := ProcessInterface;
END_SET
END_PROPERTY

PROPERTY ProcessLinkedLists : ARRAY[1..max_process] OF I_Process_LinkedList
SET
_ItfProcessList := ProcessLinkedLists;
END_SET
END_PROPERTY

PROPERTY TargetUsed : T_PROCESS
GET
TargetUsed := _wTargetUsed;
END_GET
SET
_wTargetUsed := TargetUsed;
END_SET
END_PROPERTY

END_FUNCTION_BLOCK

// ---- MAPPING/MAPPING_in.TcPOU
PROGRAM MAPPING_in
VAR
  sMapping          : STRING;
  bFirstCycle       : BOOL := TRUE;



//  TicketListOutput  : U_TICKET_LIST_DATA_OUTPUT;
//  TicketListState   : U_TICKET_LIST_STATE;
//  InstanceState     : U_INSTANCE_STATE;
//  AppState          : U_APP_STATE;
  TransportState    : U_XTS_TRANSPORT_STATE;
  StationState      : U_XTS_STATION_STATE;

  szTransportState  : ARRAY[1..2] OF UDINT;
  szAppState        : ARRAY[1..2] OF UDINT;
  szInstanceState   : ARRAY[1..2] OF UDINT;
  szTicketState     : ARRAY[1..2] OF UDINT;
  szTicketData      : ARRAY[1..2] OF UDINT;
END_VAR


IF (bFirstCycle)
THEN
  bFirstCycle         := FALSE;
  
  szTransportState [1]:= SIZEOF(TransportState);
  szTransportState [2]:= SIZEOF(GVL_XTS.XtsTransportState);
(*
  szAppState[1]       := SIZEOF(AppState);
  szAppState[2]       := SIZEOF(GVL_APPLICATION.AppState);

  szInstanceState[1]  := SIZEOF(InstanceState);
  szInstanceState[2]  := SIZEOF(GVL_APPLICATION.InstanceState);

  szTicketState[1]    := SIZEOF(TicketListState);
  szTicketState[2]    := SIZEOF(GVL_APPLICATION.TicketListState);

  szTicketData[1]     := SIZEOF(TicketListOutput);
  szTicketData[2]     := SIZEOF(GVL_APPLICATION.TicketListDataOutput);
*)
END_IF
(*
//---------------------------------------------------------------------
IF (SIZEOF(TicketListOutput) <> SIZEOF(GVL_APPLICATION.TicketListDataOutput))
THEN
  sMapping  := 'TicketListOutput sizes DO NOT match';
  RETURN;
END_IF
//---------------------------------------------------------------------
IF (SIZEOF(TicketListState) <> SIZEOF(GVL_APPLICATION.TicketListState))
THEN
  sMapping  := 'TicketListState sizes DO NOT match';
  RETURN;
END_IF
//---------------------------------------------------------------------
IF (SIZEOF(InstanceState) <> SIZEOF(GVL_APPLICATION.InstanceState))
THEN
  sMapping  := 'InstanceState sizes DO NOT match';
  RETURN;
END_IF
//---------------------------------------------------------------------
IF (SIZEOF(AppState) <> SIZEOF(GVL_APPLICATION.AppState))
THEN
  sMapping  := 'AppState sizes DO NOT match';
  RETURN;
END_IF
*)
//---------------------------------------------------------------------
IF (SIZEOF(TransportState) <> SIZEOF(GVL_XTS.XtsTransportState))
THEN
  sMapping  := 'TransportState sizes DO NOT match';
  RETURN;
END_IF
//---------------------------------------------------------------------
IF (SIZEOF(StationState) <> SIZEOF(GVL_XTS.StationState))
THEN
  sMapping  := 'StationState sizes DO NOT match';
  RETURN;
END_IF
sMapping    := 'MAPPING ACTIVE';
//-----------------------------------------------------------------------------------------
//       destination,                               source,                size
//-----------------------------------------------------------------------------------------
  memcpy(ADR(GVL_XTS.XtsTransportState),            ADR(TransportState),   SIZEOF(TransportState));
  memcpy(ADR(GVL_XTS.StationState),                 ADR(StationState),   SIZEOF(StationState));

  //memcpy(ADR(GVL_APPLICATION.AppState),             ADR(AppState),         SIZEOF(AppState));
  //GVL_APPLICATION.AppState.AppInit                  := AppSTate.stState.AppInit;

  //memcpy(ADR(GVL_APPLICATION.InstanceState),        ADR(InstanceState),    SIZEOF(InstanceState));
  //memcpy(ADR(GVL_APPLICATION.TicketListState),      ADR(TicketListState),  SIZEOF(TicketListState));
  //memcpy(ADR(GVL_APPLICATION.TicketListDataOutput), ADR(TicketListOutput), SIZEOF(TicketListOutput));
//-----------------------------------------------------------------------------------------
//-----------------------------------------------------------------------------------------

END_PROGRAM

// ---- APPLICATION/XTS_TRANSPORT_1.TcVIS
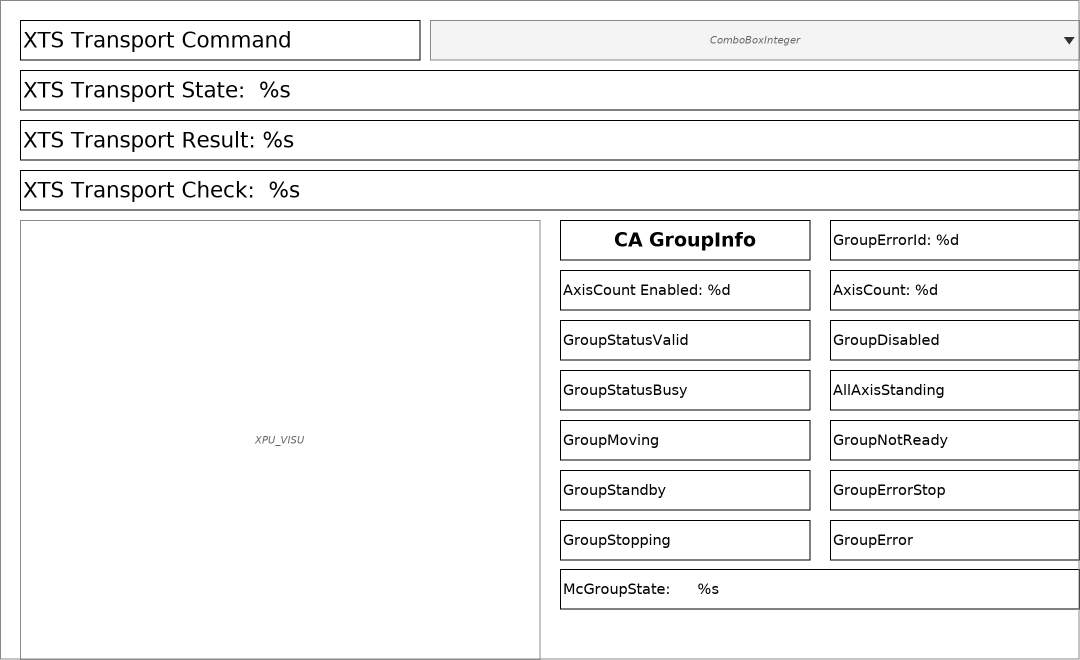
VISUALIZATION XTS_TRANSPORT_1  // 1080x660
    Rectangle (20,20 400x40), "XTS Transport Command"
    ComboBoxInteger (430,20 650x40), variable: GVL_XTS.XtsTransportCtrl.Cmd, text list: 'TL_E_CTRL_TRANSPORT'
    Rectangle (20,70 1060x40), "XTS Transport State: %s", text variable: MAIN.sTransportState
    Rectangle (20,120 1060x40), "XTS Transport Result: %s", text variable: MAIN.sTransportResult
    Rectangle (20,170 1060x40), "XTS Transport Check: %s", text variable: MAIN.sTransportCheck
    Frame (20,220 520x440)
        shows XPU_VISU(stXpuState := GVL_XTS.XtsTransportState.XpuState, stXpuInfo := GVL_XTS.XtsTransportState.XpuInfo, stXpuStrings := MAIN.stXpuStrings)
    Frame (560,220 520x390)
        shows GROUP_VISU(stGroupInfo := GVL_XTS.XtsTransportState.GroupInfo, sGroupState := MAIN.sCaGroupState)
END_VISUALIZATION

// ---- GlobalTextList.TcGTLO
TEXTLIST GlobalTextList
  17 = ' STATION_ENABLE'
  34 = ' STATION_MOVER_ENTER'
  452 = ' STATION_MOVER_GONE'
  75 = ' STATION_MOVER_OUT'
  598 = ' STATION_PROCESS_DONE'
  750 = ' STATION_PROCESS_START'
  294 = '%.2f'
  191 = '%d'
  836 = '%s'
  704 = 'All Positions Valid'
  562 = 'AllAxisStanding'
  878 = 'AxisCount Enabled: %d'
  162 = 'AxisCount: %d'
  516 = 'CA GroupInfo'
  929 = 'Control'
  707 = 'CyclicCheck: %s'
  660 = 'DC Link All Modules'
  843 = 'Detected AxisCount: %d'
  772 = 'Expected AxisCount: %d'
  48 = 'GroupDisabled'
  915 = 'GroupError'
  495 = 'GroupErrorId: %d'
  975 = 'GroupErrorStop'
  300 = 'GroupMoving'
  807 = 'GroupNotReady'
  438 = 'GroupStandby'
  226 = 'GroupStatusBusy'
  204 = 'GroupStatusValid'
  973 = 'GroupStopping'
  680 = 'ID Detection Active'
  238 = 'ID Detection Error'
  526 = 'ID Detection Mode: %s'
  29 = 'ID Detection Valid'
  211 = 'Info Act Pos Absolute'
  586 = 'Info Act Pos Modulo'
  21 = 'Info Mover Avoiding Collision'
  282 = 'Info Mover Coupled'
  398 = 'Info Mover Enabled'
  751 = 'Info Mover Error'
  907 = 'Info Mover Standstill'
  480 = 'Info nError ID'
  922 = 'Info Target Pos Absolute'
  16 = 'Info Target Pos Modulo'
  779 = 'Mask: %s'
  726 = 'McGroupState:      %s'
  974 = 'MOVER command'
  387 = 'Mover ID: %d'
  297 = 'Mover Position Assignement: %s'
  840 = 'MOVER result:  %s'
  53 = 'MOVER state:   %s'
  756 = 'nMoverSelected: %d'
  427 = 'Offset: %.3f'
  312 = 'Operation Mode: %s'
  320 = 'Queue: %d'
  91 = 'Set Acceleration'
  399 = 'Set Delta'
  382 = 'Set Distance'
  757 = 'Set Gap'
  934 = 'Set Jerk'
  201 = 'Set Override'
  936 = 'Set Position'
  62 = 'Set Velocity'
  231 = 'State'
  567 = 'Target Station: %d'
  227 = 'XpuResult:   %s'
  96 = 'XpuState:    %s'
  884 = 'XTS Station'
  572 = 'XTS Transport Check:  %s'
  500 = 'XTS Transport Command'
  395 = 'XTS Transport Result: %s'
  798 = 'XTS Transport State:  %s'
END_TEXTLIST

// ---- XTS_TRANSPORT/_Visualization/GROUP_VISU.TcVIS
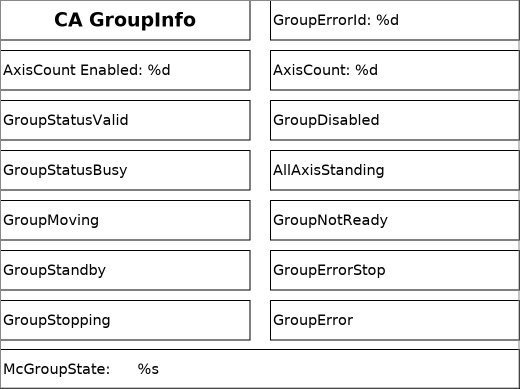
VISUALIZATION GROUP_VISU  // 520x389
VAR_IN_OUT
	stGroupInfo   : ST_GROUP_INFO;
  sGroupState   : string(60);
END_VAR
    Rectangle (0,100 250x40), "GroupStatusValid", colour toggle: stGroupInfo.GroupStatusValid
    Rectangle (0,150 250x40), "GroupStatusBusy", colour toggle: stGroupInfo.GroupStatusBusy
    Rectangle (0,200 250x40), "GroupMoving", colour toggle: stGroupInfo.GroupMoving
    Rectangle (270,250 250x40), "GroupErrorStop", colour toggle: stGroupInfo.GroupErrorStop
    Rectangle (270,200 250x40), "GroupNotReady", colour toggle: stGroupInfo.GroupNotReady
    Rectangle (0,250 250x40), "GroupStandby", colour toggle: stGroupInfo.GroupStandby
    Rectangle (0,300 250x40), "GroupStopping", colour toggle: stGroupInfo.GroupStopping
    Rectangle (270,100 250x40), "GroupDisabled", colour toggle: stGroupInfo.GroupDisabled
    Rectangle (270,150 250x40), "AllAxisStanding", colour toggle: stGroupInfo.AllAxesStanding
    Rectangle (270,300 250x40), "GroupError", colour toggle: stGroupInfo.GroupError
    Rectangle (270,0 250x40), "GroupErrorId: %d", text variable: stGroupInfo.GroupErrorId
    Rectangle (270,50 250x40), "AxisCount: %d", text variable: stGroupInfo.AxisCount
    Rectangle (0,349 520x40), "McGroupState: %s", text variable: sGroupState
    Rectangle (0,0 250x40), "CA GroupInfo"
    Rectangle (0,50 250x40), "AxisCount Enabled: %d", text variable: stGroupInfo.AxisCountEnabled
END_VISUALIZATION

